(* PLC project SWPR1010_A0_1_29.project, CODESYS CODESYS V3.5 SP16 Patch 6 *)
(* stored: creationDateTime 2025-08-05T16:58:57.5396954, modificationDateTime 2025-08-05T16:58:31.4416113 *)

TYPE BOOL_T : STRUCT
  v : BOOL := TRUE;  (* Validation Bit *)
  e : BOOL := FALSE;  (* j1939 error bit *)
  na : BOOL := FALSE;  (* j1939 not available bit *)
  x : BOOL;  (* Value Bit *)
END_STRUCT;
END_TYPE

TYPE BYTE_T : STRUCT
  v : BOOL;  (* Validation Bit *)
  e : BOOL := FALSE;  (* j1939 error bit *)
  na : BOOL := FALSE;  (* j1939 not available bit *)
  x : BYTE;  (* Value Bit *)
  J1939 : BOOL;  (* J1939 *)
  RangeExcd : BOOL;  (* Range Exceeded *)
END_STRUCT;
END_TYPE

TYPE DWORD_T : STRUCT
  v : BOOL;  (* Validation Bit *)
  e : BOOL := FALSE;  (* j1939 error bit *)
  na : BOOL := FALSE;  (* j1939 not available bit *)
  x : DWORD;  (* Value Bit *)
  J1939 : BOOL;  (* J1939 *)
  RangeExcd : BOOL;  (* Range Exceeded *)
END_STRUCT;
END_TYPE

TYPE LREAL_T : STRUCT
  v : BOOL;  (* Validation Bit *)
  e : BOOL := FALSE;  (* j1939 error bit *)
  na : BOOL := FALSE;  (* j1939 not available bit *)
  x : LREAL;  (* Value Bit *)
  J1939 : BOOL;  (* J1939 *)
  RangeExcd : BOOL;  (* Range Exceeded *)
END_STRUCT;
END_TYPE

TYPE LWORD_T : STRUCT
  v : BOOL;  (* Validation Bit *)
  e : BOOL := FALSE;  (* j1939 error bit *)
  na : BOOL := FALSE;  (* j1939 not available bit *)
  x : LWORD;  (* Value Bit *)
  J1939 : BOOL;  (* J1939 *)
  RangeExcd : BOOL;  (* Range Exceeded *)
END_STRUCT;
END_TYPE

TYPE REAL_T : STRUCT
  v : BOOL;  (* Validation Bit *)
  e : BOOL := FALSE;  (* j1939 error bit *)
  na : BOOL := FALSE;  (* j1939 not available bit *)
  x : REAL;  (* Value Bit *)
  J1939 : BOOL;  (* J1939 *)
  RangeExcd : BOOL;  (* Range Exceeded *)
END_STRUCT;
END_TYPE

TYPE UDINT_T : STRUCT
  v : BOOL;  (* Validation Bit *)
  e : BOOL := FALSE;  (* j1939 error bit *)
  na : BOOL := FALSE;  (* j1939 not available bit *)
  x : UDINT;  (* Value Bit *)
  J1939 : BOOL;  (* J1939 *)
  RangeExcd : BOOL;  (* Range Exceeded *)
END_STRUCT;
END_TYPE

TYPE UINT_T : STRUCT
  v : BOOL;  (* Validation Bit *)
  e : BOOL := FALSE;  (* j1939 error bit *)
  na : BOOL := FALSE;  (* j1939 not available bit *)
  x : UINT;  (* Value Bit *)
  J1939 : BOOL;  (* J1939 *)
  RangeExcd : BOOL;  (* Range Exceeded *)
END_STRUCT;
END_TYPE

TYPE ULINT_T : STRUCT
  v : BOOL;  (* Validation Bit *)
  e : BOOL := FALSE;  (* j1939 error bit *)
  na : BOOL := FALSE;  (* j1939 not available bit *)
  x : ULINT;  (* Value Bit *)
  J1939 : BOOL;  (* J1939 *)
  RangeExcd : BOOL;  (* Range Exceeded *)
END_STRUCT;
END_TYPE

TYPE USINT_T : STRUCT
  v : BOOL;  (* Validation Bit *)
  e : BOOL := FALSE;  (* j1939 error bit *)
  na : BOOL := FALSE;  (* j1939 not available bit *)
  x : USINT;  (* Value Bit *)
  J1939 : BOOL;  (* J1939 *)
  RangeExcd : BOOL;  (* Range Exceeded *)
END_STRUCT;
END_TYPE

TYPE WORD_T : STRUCT
  v : BOOL;  (* Validation Bit *)
  e : BOOL := FALSE;  (* j1939 error bit *)
  na : BOOL := FALSE;  (* j1939 not available bit *)
  x : WORD;  (* Value Bit *)
  J1939 : BOOL;  (* J1939 *)
  RangeExcd : BOOL;  (* Range Exceeded *)
END_STRUCT;
END_TYPE

TYPE IIVD_T : STRUCT
  X_Param_Arr : Param_T;
  X_Spd_Max : REAL_T := (v := FALSE);  (* test *)
  S_ER_Com_ECU : BOOL_T := (v := FALSE);  (* ****************************************** MESSAGE: Haberlesme_Durumlari ID: 200 ****************************************** S_ER_Com_ECU/StartBit:0/Length:2/J1939:YES *)
  S_ER_Com_DWP_ICAN : BOOL_T := (v := FALSE);  (* S_ER_Com_DWP_ICAN/StartBit:2/Length:2/J1939:YES *)
  S_ER_Com_DWP_XCAN : BOOL_T := (v := FALSE);  (* S_ER_Com_DWP_XCAN/StartBit:4/Length:2/J1939:YES *)
  S_ER_Com_Str_Pmp : BOOL_T := (v := FALSE);  (* S_ER_Com_Str_Pmp/StartBit:6/Length:2/J1939:YES *)
  S_ER_Com_Fus_Chk_ID0 : BOOL_T := (v := FALSE);  (* S_ER_Com_Fus_Chk_ID0/StartBit:8/Length:2/J1939:YES *)
  S_ER_Com_Fus_Chk_ID1 : BOOL_T := (v := FALSE);  (* S_ER_Com_Fus_Chk_ID1/StartBit:10/Length:2/J1939:YES *)
  S_ER_Com_Fus_Chk_ID2 : BOOL_T := (v := FALSE);  (* S_ER_Com_Fus_Chk_ID2/StartBit:12/Length:2/J1939:YES *)
  S_ER_Com_ECAS : BOOL_T := (v := FALSE);  (* S_ER_Com_ECAS/StartBit:14/Length:2/J1939:YES *)
  S_ER_Com_Snd_Gen : BOOL_T := (v := FALSE);  (* S_ER_Com_Snd_Gen/StartBit:16/Length:2/J1939:YES *)
  S_ER_Com_DCAN : BOOL_T := (v := FALSE);  (* S_ER_Com_DCAN/StartBit:18/Length:2/J1939:YES *)
  S_ER_Com_Node1 : BOOL_T := (v := FALSE);  (* S_ER_Com_Node1/StartBit:24/Length:2/J1939:YES *)
  S_ER_Com_Node2 : BOOL_T := (v := FALSE);  (* S_ER_Com_Node2/StartBit:26/Length:2/J1939:YES *)
  S_ER_Com_Node3 : BOOL_T := (v := FALSE);  (* S_ER_Com_Node3/StartBit:28/Length:2/J1939:YES *)
  S_ER_Com_Node4 : BOOL_T := (v := FALSE);  (* S_ER_Com_Node4/StartBit:30/Length:2/J1939:YES *)
  S_ER_Com_Node5 : BOOL_T := (v := FALSE);  (* S_ER_Com_Node5/StartBit:32/Length:2/J1939:YES *)
  S_ER_Com_Node6 : BOOL_T := (v := FALSE);  (* S_ER_Com_Node6/StartBit:34/Length:2/J1939:YES *)
  S_ER_Com_Node8 : BOOL_T := (v := FALSE);  (* S_ER_Com_Node8/StartBit:38/Length:2/J1939:YES *)
  S_ER_Com_Dr1 : BOOL_T := (v := FALSE);  (* S_ER_Com_Dr1/StartBit:40/Length:2/J1939:YES *)
  S_ER_Com_Dr2 : BOOL_T := (v := FALSE);  (* S_ER_Com_Dr2/StartBit:42/Length:2/J1939:YES *)
  S_ER_Com_Dr3 : BOOL_T := (v := FALSE);  (* S_ER_Com_Dr3/StartBit:44/Length:2/J1939:YES *)
  S_ER_Com_Dr4 : BOOL_T := (v := FALSE);  (* S_ER_Com_Dr4/StartBit:46/Length:2/J1939:YES *)
  S_ER_Com_Dr5 : BOOL_T := (v := FALSE);  (* S_ER_Com_Dr5/StartBit:48/Length:2/J1939:YES *)
  S_ER_Com_Dr6 : BOOL_T := (v := FALSE);  (* S_ER_Com_Dr6/StartBit:50/Length:2/J1939:YES *)
  S_ER_Com_Dr7 : BOOL_T := (v := FALSE);  (* S_ER_Com_Dr7/StartBit:52/Length:2/J1939:YES *)
  S_ER_Com_Dr8 : BOOL_T := (v := FALSE);  (* S_ER_Com_Dr8/StartBit:54/Length:2/J1939:YES *)
  S_ER_Com_Dr9 : BOOL_T := (v := FALSE);  (* S_ER_Com_Dr9/StartBit:56/Length:2/J1939:YES *)
  S_Warn_Knl_Mn_Cond : BOOL_T := (v := FALSE);  (* S_Warn_Knl_Mn_Cond/StartBit:58/Length:2/J1939:YES *)
  S_ER_Lmp_Oc : BOOL_T := (v := FALSE);  (* S_ER_Lmp_Oc/StartBit:60/Length:2/J1939:YES *)
  S_ER_Mir_Windw_Heat_En : BOOL_T := (v := FALSE);  (* S_ER_Mir_Windw_Heat_En/StartBit:62/Length:2/J1939:YES *)
  W_Str_Pmp_Spd : REAL_T := (v := FALSE);  (* ****************************************** MESSAGE: Direksiyon_Pompasi_Analog ID: 210 ****************************************** W_Str_Pmp_Spd/StartBit:0/Length:16/J1939:YES *)
  X_Str_Pmp_Spd : REAL_T := (v := FALSE);  (* X_Str_Pmp_Spd/StartBit:16/Length:16/J1939:YES *)
  X_P_Str_Pmp : REAL_T := (v := FALSE);  (* X_P_Str_Pmp/StartBit:32/Length:16/J1939:YES *)
  X_I_Str_Pmp : REAL_T := (v := FALSE);  (* X_I_Str_Pmp/StartBit:48/Length:9/J1939:NO *)
  C_Str_Pmp_En : BOOL_T := (v := FALSE);  (* ****************************************** MESSAGE: Direksiyon_Pompasi_Durum ID: 211 ****************************************** C_Str_Pmp_En/StartBit:0/Length:2/J1939:YES *)
  S_Str_Pmp_Em_Run_FOC : BOOL_T := (v := FALSE);  (* S_Str_Pmp_Em_Run_FOC/StartBit:2/Length:2/J1939:YES *)
  S_Str_Pmp_Em_Run_Slp : BOOL_T := (v := FALSE);  (* S_Str_Pmp_Em_Run_Slp/StartBit:4/Length:2/J1939:YES *)
  S_ER_Str_Pmp : BOOL_T := (v := FALSE);  (* S_ER_Str_Pmp/StartBit:6/Length:2/J1939:YES *)
  S_Str_Pmp_Run : BOOL_T := (v := FALSE);  (* S_Str_Pmp_Run/StartBit:8/Length:2/J1939:YES *)
  X_T_Str_Pmp_Mot : REAL_T := (v := FALSE);  (* X_T_Str_Pmp_Mot/StartBit:16/Length:8/J1939:YES *)
  X_T_Str_Pmp_Inver : REAL_T := (v := FALSE);  (* X_T_Str_Pmp_Inver/StartBit:24/Length:8/J1939:YES *)
  X_Mot_Load_Str_Pmp : REAL_T := (v := FALSE);  (* X_Mot_Load_Str_Pmp/StartBit:32/Length:8/J1939:YES *)
  X_T_Air_Cmp : REAL_T := (v := FALSE);  (* X_T_Air_Cmp/StartBit:48/Length:8/J1939:YES *)
  S_ER_Air_Cmp_Tmp : BOOL_T := (v := FALSE);  (* S_ER_Air_Cmp_Tmp/StartBit:56/Length:2/J1939:YES *)
  S_Air_Cmp_Filt_Warn_Actv : BOOL_T := (v := FALSE);  (* S_Air_Cmp_Filt_Warn_Actv/StartBit:58/Length:2/J1939:YES *)
  S_Hld_Brk_Byp : BOOL_T := (v := FALSE);  (* ****************************************** MESSAGE: Arac_Durumlari ID: 220 ****************************************** S_Hld_Brk_Byp/StartBit:0/Length:2/J1939:YES *)
  S_Hld_Brk_Req : BOOL_T := (v := FALSE);  (* S_Hld_Brk_Req/StartBit:2/Length:2/J1939:YES *)
  S_Hld_Brk_Actv : BOOL_T := (v := FALSE);  (* S_Hld_Brk_Actv/StartBit:4/Length:2/J1939:YES *)
  S_Aut_Lub_Oil_Lv_Lo : BOOL_T := (v := FALSE);  (* S_Aut_Lub_Oil_Lv_Lo/StartBit:6/Length:2/J1939:YES *)
  S_ECAS_Dwn_Req : BOOL_T := (v := FALSE);  (* S_ECAS_Dwn_Req/StartBit:8/Length:2/J1939:YES *)
  S_ECAS_Up_Req : BOOL_T := (v := FALSE);  (* S_ECAS_Up_Req/StartBit:10/Length:2/J1939:YES *)
  S_ECAS_Pos_Down : BOOL_T := (v := FALSE);  (* S_ECAS_Pos_Down/StartBit:12/Length:2/J1939:YES *)
  S_ECAS_Pos_Up : BOOL_T := (v := FALSE);  (* S_ECAS_Pos_Up/StartBit:14/Length:2/J1939:YES *)
  S_Knl_Req : BOOL_T := (v := FALSE);  (* S_Knl_Req/StartBit:16/Length:2/J1939:YES *)
  S_Knl_Actv : BOOL_T := (v := FALSE);  (* S_Knl_Actv/StartBit:18/Length:2/J1939:YES *)
  S_Fwd_Gear : BOOL_T := (v := FALSE);  (* S_Fwd_Gear/StartBit:20/Length:2/J1939:YES *)
  S_Bwd_Gear : BOOL_T := (v := FALSE);  (* S_Bwd_Gear/StartBit:22/Length:2/J1939:YES *)
  S_Vh_Actv_Key_Lv1 : BOOL_T := (v := FALSE);  (* S_Vh_Actv_Key_Lv1/StartBit:24/Length:2/J1939:YES *)
  S_Vh_Actv_Key_Lv2 : BOOL_T := (v := FALSE);  (* S_Vh_Actv_Key_Lv2/StartBit:26/Length:2/J1939:YES *)
  S_Vh_Actv_Key_Lv3 : BOOL_T := (v := FALSE);  (* S_Vh_Actv_Key_Lv3/StartBit:28/Length:2/J1939:YES *)
  S_Brk_Park : BOOL_T := (v := FALSE);  (* S_Brk_Park/StartBit:30/Length:2/J1939:YES *)
  Z_Ret_Lv : BYTE_T := (v := FALSE);  (* Z_Ret_Lv/StartBit:32/Length:4/J1939:YES *)
  S_Aut_Lub_Actv : BOOL_T := (v := FALSE);  (* S_Aut_Lub_Actv/StartBit:36/Length:2/J1939:YES *)
  S_ER_Aut_Lub_Snsr : BOOL_T := (v := FALSE);  (* S_ER_Aut_Lub_Snsr/StartBit:38/Length:2/J1939:YES *)
  S_Bat_Mod_Btn : BOOL_T := (v := FALSE);  (* S_Bat_Mod_Btn/StartBit:42/Length:2/J1939:YES *)
  S_Elec_Mod_Btn : BOOL_T := (v := FALSE);  (* S_Elec_Mod_Btn/StartBit:44/Length:2/J1939:YES *)
  S_Bwd_Lft_Chrg_Btn : BOOL_T := (v := FALSE);  (* S_Bwd_Lft_Chrg_Btn/StartBit:12/Length:2/J1939:YES *)
  S_Bwd_Lft_Chrg_Em_Stop_Swc1 : BOOL_T := (v := FALSE);  (* S_Bwd_Lft_Chrg_Em_Stop_Swc1/StartBit:14/Length:2/J1939:YES *)
  S_Bwd_Lft_Chrg_Em_Stop_Swc2 : BOOL_T := (v := FALSE);  (* S_Bwd_Lft_Chrg_Em_Stop_Swc2/StartBit:16/Length:2/J1939:YES *)
  Z_Config_Clu : BYTE_T := (v := FALSE);  (* Z_Config_Clu/StartBit:56/Length:8/J1939:YES *)
  X_Axl1_Brk_Ling_1 : REAL_T := (v := FALSE);  (* ****************************************** MESSAGE: Fren_balata_durumlari ID: 221 ****************************************** X_Axl1_Brk_Ling_1/StartBit:0/Length:8/J1939:YES *)
  X_Axl1_Brk_Ling_2 : REAL_T := (v := FALSE);  (* X_Axl1_Brk_Ling_2/StartBit:8/Length:8/J1939:YES *)
  X_Axl2_Brk_Ling_1 : REAL_T := (v := FALSE);  (* X_Axl2_Brk_Ling_1/StartBit:16/Length:8/J1939:YES *)
  X_Axl2_Brk_Ling_2 : REAL_T := (v := FALSE);  (* X_Axl2_Brk_Ling_2/StartBit:24/Length:8/J1939:YES *)
  X_Axl3_Brk_Ling_1 : REAL_T := (v := FALSE);  (* X_Axl3_Brk_Ling_1/StartBit:32/Length:8/J1939:YES *)
  X_Axl3_Brk_Ling_2 : REAL_T := (v := FALSE);  (* X_Axl3_Brk_Ling_2/StartBit:40/Length:8/J1939:YES *)
  X_Axl4_Brk_Ling_1 : REAL_T := (v := FALSE);  (* X_Axl4_Brk_Ling_1/StartBit:48/Length:8/J1939:YES *)
  X_Axl4_Brk_Ling_2 : REAL_T := (v := FALSE);  (* X_Axl4_Brk_Ling_2/StartBit:56/Length:8/J1939:YES *)
  S_ER_Not_Ins_Pr_Sns_Frnt_Brk : BOOL_T := (v := FALSE);  (* ****************************************** MESSAGE: Fren_Basinclari ID: 222 ****************************************** S_ER_Not_Ins_Pr_Sns_Frnt_Brk/StartBit:0/Length:2/J1939:YES *)
  S_ER_Not_Ins_Pr_Sns_Bwd_Brk : BOOL_T := (v := FALSE);  (* S_ER_Not_Ins_Pr_Sns_Bwd_Brk/StartBit:2/Length:2/J1939:YES *)
  S_ER_Not_Ins_Pr_Snsr_Prk_Brk : BOOL_T := (v := FALSE);  (* S_ER_Not_Ins_Pr_Snsr_Prk_Brk/StartBit:4/Length:2/J1939:YES *)
  S_ER_Not_Ins_Pr_Sns_Susp_Rr : BOOL_T := (v := FALSE);  (* S_ER_Not_Ins_Pr_Sns_Susp/StartBit:6/Length:2/J1939:YES *)
  S_ER_Not_Ins_Pr_Sns_Susp_Frnt : BOOL_T := (v := FALSE);  (* S_ER_Not_Ins_Pr_Sns_Susp_Frnt/StartBit:8/Length:2/J1939:YES *)
  S_ER_Brk_Lnng : BOOL_T := (v := FALSE);  (* S_ER_Brk_Lnng/StartBit:8/Length:2/J1939:YES *)
  S_ER_Pin_Pr_Air : BOOL_T := (v := FALSE);  (* S_ER_Pin_Pr_Air/StartBit:12/Length:2/J1939:YES *)
  X_Pr_Air_Tank_Brk_Bwd : REAL_T := (v := FALSE);  (* X_Pr_Air_Tank_Brk_Bwd/StartBit:16/Length:8/J1939:YES *)
  X_Pr_Air_Tank_Brk_Frnt : REAL_T := (v := FALSE);  (* X_Pr_Air_Tank_Brk_Frnt/StartBit:24/Length:8/J1939:YES *)
  X_Pr_Air_Tank_Brk_Prk : REAL_T := (v := FALSE);  (* X_Pr_Air_Tank_Brk_Prk/StartBit:32/Length:8/J1939:YES *)
  X_Pr_Air_Tank_Susp_Rr : REAL_T := (v := FALSE);  (* X_Pr_Air_Tank_Susp_Rr/StartBit:40/Length:8/J1939:YES *)
  X_Pr_Air_Tank_Susp_Frnt : REAL_T := (v := FALSE);  (* X_Pr_Air_Tank_Susp_Frnt/StartBit:48/Length:8/J1939:YES *)
  X_Pr_Axl1_Wh1 : REAL_T := (v := FALSE);  (* ****************************************** MESSAGE: Lastik_Basinclari_1 ID: 223 ****************************************** X_Pr_Axl1_Wh1/StartBit:0/Length:8/J1939:YES *)
  X_Pr_Axl1_Wh2 : REAL_T := (v := FALSE);  (* X_Pr_Axl1_Wh2/StartBit:8/Length:8/J1939:YES *)
  X_Pr_Axl2_Wh1 : REAL_T := (v := FALSE);  (* X_Pr_Axl2_Wh1/StartBit:16/Length:8/J1939:YES *)
  X_Pr_Axl2_Wh2 : REAL_T := (v := FALSE);  (* X_Pr_Axl2_Wh2/StartBit:24/Length:8/J1939:YES *)
  X_Pr_Axl2_Wh3 : REAL_T := (v := FALSE);  (* X_Pr_Axl2_Wh3/StartBit:32/Length:8/J1939:YES *)
  X_Pr_Axl2_Wh4 : REAL_T := (v := FALSE);  (* X_Pr_Axl2_Wh4/StartBit:40/Length:8/J1939:YES *)
  X_Pr_Axl3_Wh1 : REAL_T := (v := FALSE);  (* ****************************************** MESSAGE: Lastik_Basinclari_2 ID: 224 ****************************************** X_Pr_Axl3_Wh1/StartBit:0/Length:8/J1939:YES *)
  X_Pr_Axl3_Wh2 : REAL_T := (v := FALSE);  (* X_Pr_Axl3_Wh2/StartBit:8/Length:8/J1939:YES *)
  X_Pr_Axl3_Wh3 : REAL_T := (v := FALSE);  (* X_Pr_Axl3_Wh3/StartBit:16/Length:8/J1939:YES *)
  X_Pr_Axl3_Wh4 : REAL_T := (v := FALSE);  (* X_Pr_Axl3_Wh4/StartBit:24/Length:8/J1939:YES *)
  X_Pr_Axl4_Wh1 : REAL_T := (v := FALSE);  (* X_Pr_Axl4_Wh1/StartBit:32/Length:8/J1939:YES *)
  X_Pr_Axl4_Wh2 : REAL_T := (v := FALSE);  (* X_Pr_Axl4_Wh2/StartBit:40/Length:8/J1939:YES *)
  X_Pr_Axl4_Wh3 : REAL_T := (v := FALSE);  (* X_Pr_Axl4_Wh3/StartBit:48/Length:8/J1939:YES *)
  X_Pr_Axl4_Wh4 : REAL_T := (v := FALSE);  (* X_Pr_Axl4_Wh4/StartBit:56/Length:8/J1939:YES *)
  S_Cvr_Op_Dr1_Ext : BOOL_T := (v := FALSE);  (* ****************************************** MESSAGE: Arac_Bilgilendirme ID: 225 ****************************************** S_Cvr_Op_Dr1_Ext/StartBit:0/Length:2/J1939:YES *)
  S_Cvr_Op_Lic : BOOL_T := (v := FALSE);  (* S_Cvr_Op_Lic/StartBit:2/Length:2/J1939:YES *)
  S_Cvr_Op_Bat_Room : BOOL_T := (v := FALSE);  (* S_Cvr_Op_Bat_Room/StartBit:4/Length:2/J1939:YES *)
  S_Cvr_Op_Mot : BOOL_T := (v := FALSE);  (* S_Cvr_Op_Mot/StartBit:10/Length:2/J1939:YES *)
  S_Cvr_Op_Bwd_Lft_Chrg : BOOL_T := (v := FALSE);  (* S_Cvr_Op_Bwd_Lft_Chrg/StartBit:12/Length:2/J1939:YES *)
  S_Cvr_Op_24V_Chrg_Plg : BOOL_T := (v := FALSE);  (* S_Cvr_Op_24V_Chrg_Plg/StartBit:14/Length:2/J1939:YES *)
  S_Cvr_Op_Bwd : BOOL_T := (v := FALSE);  (* S_Cvr_Op_Bwd/StartBit:16/Length:2/J1939:YES *)
  S_Rp_Op : BOOL_T := (v := FALSE);  (* S_Rp_Op/StartBit:18/Length:2/J1939:YES *)
  S_Cvr_Op_Bwd_Mnt_Pnl : BOOL_T := (v := FALSE);  (* S_Cvr_Op_Bwd_Mnt_Pnl/StartBit:20/Length:2/J1939:YES *)
  S_Cvr_Op_Frnt_Mnt_Pnl : BOOL_T := (v := FALSE);  (* S_Cvr_Op_Frnt_Mnt_Pnl/StartBit:22/Length:2/J1939:YES *)
  S_ER_Rp_Op_Unauth : BOOL_T := (v := FALSE);  (* S_ER_Rp_Op_Unauth/StartBit:30/Length:2/J1939:YES *)
  S_ER_Fi_Bat_Room : BOOL_T := (v := FALSE);  (* S_ER_Fi_Bat_Room/StartBit:32/Length:2/J1939:YES *)
  S_ER_Not_Ins_Fi_Sens_Bat_Room : BOOL_T := (v := FALSE);  (* S_ER_Not_Ins_Fi_Sens_Bat_Room/StartBit:34/Length:2/J1939:YES *)
  S_ER_Fi_Frnt_Pnl : BOOL_T := (v := FALSE);  (* S_ER_Fi_Frnt_Pnl/StartBit:36/Length:2/J1939:YES *)
  S_ER_Not_Ins_Fi_Snsr_Frnt_Pnl : BOOL_T := (v := FALSE);  (* S_ER_Not_Ins_Fi_Snsr_Frnt_Pnl/StartBit:38/Length:2/J1939:YES *)
  S_ER_Fi_Drv_Mot : BOOL_T := (v := FALSE);  (* S_ER_Fi_Drv_Mot/StartBit:40/Length:2/J1939:YES *)
  S_ER_Not_Ins_Fi_Snsr_Drv_Mot : BOOL_T := (v := FALSE);  (* S_ER_Not_Ins_Fi_Snsr_Drv_Mot/StartBit:42/Length:2/J1939:YES *)
  S_ER_Fi_Bwd_Pnl : BOOL_T := (v := FALSE);  (* S_ER_Fi_Bwd_Pnl/StartBit:44/Length:2/J1939:YES *)
  S_ER_Not_Ins_Fi_Snsr_Bwd_Pnl : BOOL_T := (v := FALSE);  (* S_ER_Not_Ins_Fi_Snsr_Bwd_Pnl/StartBit:46/Length:2/J1939:YES *)
  S_ER_Fi_Eng_Room : BOOL_T := (v := FALSE);  (* S_ER_Fi_Eng_Room/StartBit:48/Length:2/J1939:YES *)
  S_ER_Not_Ins_Fi_Sns_Eng_Room : BOOL_T := (v := FALSE);  (* S_ER_Not_Ins_Fi_Sns_Eng_Room/StartBit:50/Length:2/J1939:YES *)
  X_Psng_No : REAL_T := (v := FALSE);  (* ****************************************** MESSAGE: Arac_Kritik_Uyarilari ID: 226 ****************************************** X_Psng_No/StartBit:0/Length:8/J1939:YES *)
  X_Wgt_Axle : REAL_T := (v := FALSE);  (* X_Wgt_Axle/StartBit:8/Length:16/J1939:YES *)
  C_Err_Pg_Dn : BOOL_T := (v := FALSE);  (* C_Err_Pg_Dn/StartBit:24/Length:2/J1939:YES *)
  C_Err_Pg_Up : BOOL_T := (v := FALSE);  (* C_Err_Pg_Up/StartBit:26/Length:2/J1939:YES *)
  C_Rst_Trip : BOOL_T := (v := FALSE);  (* C_Rst_Trip/StartBit:28/Length:2/J1939:YES *)
  S_Drug_Alch_Ctrl : BOOL_T := (v := FALSE);  (* S_Drug_Alch_Ctrl/StartBit:32/Length:2/J1939:YES *)
  S_Drug_Alch_Warn : BOOL_T := (v := FALSE);  (* S_Drug_Alch_Warn/StartBit:34/Length:2/J1939:YES *)
  S_Prheat_Tk_Lv_Lo : BOOL_T := (v := FALSE);  (* C_Flr_Heat_Off/StartBit:36/Length:2/J1939:YES *)
  S_ER_Wpr_Wtr_Lv : BOOL_T := (v := FALSE);  (* S_ER_Wpr_Wtr_Lv/StartBit:40/Length:2/J1939:YES *)
  S_Sfty_Belt_Ins : BOOL_T := (v := FALSE);  (* S_Sfty_Belt_Ins/StartBit:42/Length:2/J1939:YES *)
  C_Pnt_Up : BOOL_T := (v := FALSE);  (* C_Pnt_Up/StartBit:44/Length:2/J1939:YES *)
  C_Pnt_Dn : BOOL_T := (v := FALSE);  (* C_Pnt_Dn/StartBit:46/Length:2/J1939:YES *)
  S_Drv_Seat_Pre_Snsr : BOOL_T := (v := FALSE);  (* S_Drv_Seat_Pre_Snsr/StartBit:48/Length:2/J1939:YES *)
  S_Inc_Acc : BOOL_T := (v := FALSE);  (* S_Inc_Acc/StartBit:56/Length:2/J1939:YES *)
  S_Inc_Stop : BOOL_T := (v := FALSE);  (* S_Inc_Stop/StartBit:58/Length:2/J1939:YES *)
  S_Er_Tire_Pres : BOOL_T := (v := FALSE);  (* S_Er_Tire_Pres/StartBit:60/Length:2/J1939:YES *)
  Z_Dr1_Err_Fram_1 : BYTE_T := (v := FALSE);  (* ****************************************** MESSAGE: Kapi_Hatalari_1 ID: 230 ****************************************** Z_Dr1_Err_Fram_1/StartBit:0/Length:8/J1939:YES *)
  Z_Dr1_Err_Fram_2 : BYTE_T := (v := FALSE);  (* Z_Dr1_Err_Fram_2/StartBit:8/Length:8/J1939:YES *)
  Z_Dr1_Err_Fram_3 : BYTE_T := (v := FALSE);  (* Z_Dr1_Err_Fram_3/StartBit:16/Length:8/J1939:YES *)
  Z_Dr2_Err_Fram_1 : BYTE_T := (v := FALSE);  (* Z_Dr2_Err_Fram_1/StartBit:32/Length:8/J1939:YES *)
  Z_Dr2_Err_Fram_2 : BYTE_T := (v := FALSE);  (* Z_Dr2_Err_Fram_2/StartBit:40/Length:8/J1939:YES *)
  Z_Dr2_Err_Fram_3 : BYTE_T := (v := FALSE);  (* Z_Dr2_Err_Fram_3/StartBit:48/Length:8/J1939:YES *)
  Z_Dr3_Err_Fram_1 : BYTE_T := (v := FALSE);  (* ****************************************** MESSAGE: Kapi_Hatalari_2 ID: 231 ****************************************** Z_Dr3_Err_Fram_1/StartBit:0/Length:8/J1939:YES *)
  Z_Dr3_Err_Fram_2 : BYTE_T := (v := FALSE);  (* Z_Dr3_Err_Fram_2/StartBit:8/Length:8/J1939:YES *)
  Z_Dr3_Err_Fram_3 : BYTE_T := (v := FALSE);  (* Z_Dr3_Err_Fram_3/StartBit:16/Length:8/J1939:YES *)
  Z_Dr4_Err_Fram_1 : BYTE_T := (v := FALSE);  (* Z_Dr4_Err_Fram_1/StartBit:32/Length:8/J1939:YES *)
  Z_Dr4_Err_Fram_2 : BYTE_T := (v := FALSE);  (* Z_Dr4_Err_Fram_2/StartBit:40/Length:8/J1939:YES *)
  Z_Dr4_Err_Fram_3 : BYTE_T := (v := FALSE);  (* Z_Dr4_Err_Fram_3/StartBit:48/Length:8/J1939:YES *)
  Z_Dr5_Err_Fram_1 : BYTE_T := (v := FALSE);  (* ****************************************** MESSAGE: Kapi_Hatalari_3 ID: 232 ****************************************** Z_Dr5_Err_Fram_1/StartBit:0/Length:8/J1939:YES *)
  Z_Dr5_Err_Fram_2 : BYTE_T := (v := FALSE);  (* Z_Dr5_Err_Fram_2/StartBit:8/Length:8/J1939:YES *)
  Z_Dr5_Err_Fram_3 : BYTE_T := (v := FALSE);  (* Z_Dr5_Err_Fram_3/StartBit:16/Length:8/J1939:YES *)
  Z_Dr6_Err_Fram_1 : BYTE_T := (v := FALSE);  (* Z_Dr6_Err_Fram_1/StartBit:32/Length:8/J1939:YES *)
  Z_Dr6_Err_Fram_2 : BYTE_T := (v := FALSE);  (* Z_Dr6_Err_Fram_2/StartBit:40/Length:8/J1939:YES *)
  Z_Dr6_Err_Fram_3 : BYTE_T := (v := FALSE);  (* Z_Dr6_Err_Fram_3/StartBit:48/Length:8/J1939:YES *)
  Z_Dr7_Err_Fram_1 : BYTE_T := (v := FALSE);  (* ****************************************** MESSAGE: Kapi_Hatalari_4 ID: 233 ****************************************** Z_Dr7_Err_Fram_1/StartBit:0/Length:8/J1939:YES *)
  Z_Dr7_Err_Fram_2 : BYTE_T := (v := FALSE);  (* Z_Dr7_Err_Fram_2/StartBit:8/Length:8/J1939:YES *)
  Z_Dr7_Err_Fram_3 : BYTE_T := (v := FALSE);  (* Z_Dr7_Err_Fram_3/StartBit:16/Length:8/J1939:YES *)
  Z_Dr8_Err_Fram_1 : BYTE_T := (v := FALSE);  (* Z_Dr8_Err_Fram_1/StartBit:32/Length:8/J1939:YES *)
  Z_Dr8_Err_Fram_2 : BYTE_T := (v := FALSE);  (* Z_Dr8_Err_Fram_2/StartBit:40/Length:8/J1939:YES *)
  Z_Dr8_Err_Fram_3 : BYTE_T := (v := FALSE);  (* Z_Dr8_Err_Fram_3/StartBit:48/Length:8/J1939:YES *)
  Z_Dr9_Err_Fram_1 : BYTE_T := (v := FALSE);  (* ****************************************** MESSAGE: Kapi_Hatalari_5 ID: 234 ****************************************** Z_Dr9_Err_Fram_1/StartBit:0/Length:8/J1939:YES *)
  Z_Dr9_Err_Fram_2 : BYTE_T := (v := FALSE);  (* Z_Dr9_Err_Fram_2/StartBit:8/Length:8/J1939:YES *)
  Z_Dr9_Err_Fram_3 : BYTE_T := (v := FALSE);  (* Z_Dr9_Err_Fram_3/StartBit:16/Length:8/J1939:YES *)
  S_Dr1_Rhs_Leaf_Opng : BOOL_T := (v := FALSE);  (* ****************************************** MESSAGE: Kapi_Durum_1 ID: 235 ****************************************** S_Dr1_Rhs_Leaf_Opng/StartBit:0/Length:2/J1939:YES *)
  S_Dr1_Rhs_Leaf_Clng : BOOL_T := (v := FALSE);  (* S_Dr1_Rhs_Leaf_Clng/StartBit:2/Length:2/J1939:YES *)
  S_Dr1_Rhs_Leaf_Op : BOOL_T := (v := FALSE);  (* S_Dr1_Rhs_Leaf_Op/StartBit:4/Length:2/J1939:YES *)
  S_Dr1_Rhs_Leaf_Cl : BOOL_T := (v := FALSE);  (* S_Dr1_Rhs_Leaf_Cl/StartBit:6/Length:2/J1939:YES *)
  S_Dr1_Rhs_Leaf_Obs : BOOL_T := (v := FALSE);  (* S_Dr1_Rhs_Leaf_Obs/StartBit:8/Length:2/J1939:YES *)
  S_Dr1_Lft_Leaf_Opng : BOOL_T := (v := FALSE);  (* S_Dr1_Lft_Leaf_Opng/StartBit:10/Length:2/J1939:YES *)
  S_Dr1_Lft_Leaf_Clng : BOOL_T := (v := FALSE);  (* S_Dr1_Lft_Leaf_Clng/StartBit:12/Length:2/J1939:YES *)
  S_Dr1_Lft_Leaf_Op : BOOL_T := (v := FALSE);  (* S_Dr1_Lft_Leaf_Op/StartBit:14/Length:2/J1939:YES *)
  S_Dr1_Lft_Leaf_Cl : BOOL_T := (v := FALSE);  (* S_Dr1_Lft_Leaf_Cl/StartBit:16/Length:2/J1939:YES *)
  S_Dr1_Lft_Leaf_Obs : BOOL_T := (v := FALSE);  (* S_Dr1_Lft_Leaf_Obs/StartBit:18/Length:2/J1939:YES *)
  S_Dr1_Em_Swc : BOOL_T := (v := FALSE);  (* S_Dr1_Em_Swc/StartBit:20/Length:2/J1939:YES *)
  S_Dr2_Opng : BOOL_T := (v := FALSE);  (* S_Dr2_Opng/StartBit:24/Length:2/J1939:YES *)
  S_Dr2_Clng : BOOL_T := (v := FALSE);  (* S_Dr2_Clng/StartBit:26/Length:2/J1939:YES *)
  S_Dr2_Op : BOOL_T := (v := FALSE);  (* S_Dr2_Op/StartBit:28/Length:2/J1939:YES *)
  S_Dr2_Cl : BOOL_T := (v := FALSE);  (* S_Dr2_Cl/StartBit:30/Length:2/J1939:YES *)
  S_Dr2_Obs : BOOL_T := (v := FALSE);  (* S_Dr2_Obs/StartBit:32/Length:2/J1939:YES *)
  S_Dr2_Em_Swc : BOOL_T := (v := FALSE);  (* S_Dr2_Em_Swc/StartBit:34/Length:2/J1939:YES *)
  S_Dr3_Opng : BOOL_T := (v := FALSE);  (* S_Dr3_Opng/StartBit:40/Length:2/J1939:YES *)
  S_Dr3_Clng : BOOL_T := (v := FALSE);  (* S_Dr3_Clng/StartBit:42/Length:2/J1939:YES *)
  S_Dr3_Op : BOOL_T := (v := FALSE);  (* S_Dr3_Op/StartBit:44/Length:2/J1939:YES *)
  S_Dr3_Cl : BOOL_T := (v := FALSE);  (* S_Dr3_Cl/StartBit:46/Length:2/J1939:YES *)
  S_Dr3_Obs : BOOL_T := (v := FALSE);  (* S_Dr3_Obs/StartBit:48/Length:2/J1939:YES *)
  S_Dr3_Em_Swc : BOOL_T := (v := FALSE);  (* S_Dr3_Em_Swc/StartBit:50/Length:2/J1939:YES *)
  S_Dr4_Opng : BOOL_T := (v := FALSE);  (* ****************************************** MESSAGE: Kapi_Durum_2 ID: 237 ****************************************** S_Dr4_Opng/StartBit:0/Length:2/J1939:YES *)
  S_Dr4_Clng : BOOL_T := (v := FALSE);  (* S_Dr4_Clng/StartBit:2/Length:2/J1939:YES *)
  S_Dr4_Op : BOOL_T := (v := FALSE);  (* S_Dr4_Op/StartBit:4/Length:2/J1939:YES *)
  S_Dr4_Cl : BOOL_T := (v := FALSE);  (* S_Dr4_Cl/StartBit:6/Length:2/J1939:YES *)
  S_Dr4_Obs : BOOL_T := (v := FALSE);  (* S_Dr4_Obs/StartBit:8/Length:2/J1939:YES *)
  S_Dr4_Em_Swc : BOOL_T := (v := FALSE);  (* S_Dr4_Em_Swc/StartBit:10/Length:2/J1939:YES *)
  S_Dr5_Opng : BOOL_T := (v := FALSE);  (* S_Dr5_Opng/StartBit:16/Length:2/J1939:YES *)
  S_Dr5_Clng : BOOL_T := (v := FALSE);  (* S_Dr5_Clng/StartBit:18/Length:2/J1939:YES *)
  S_Dr5_Op : BOOL_T := (v := FALSE);  (* S_Dr5_Op/StartBit:20/Length:2/J1939:YES *)
  S_Dr5_Cl : BOOL_T := (v := FALSE);  (* S_Dr5_Cl/StartBit:22/Length:2/J1939:YES *)
  S_Dr5_Obs : BOOL_T := (v := FALSE);  (* S_Dr5_Obs/StartBit:24/Length:2/J1939:YES *)
  S_Dr5_Em_Swc : BOOL_T := (v := FALSE);  (* S_Dr5_Em_Swc/StartBit:26/Length:2/J1939:YES *)
  S_Dr6_Opng : BOOL_T := (v := FALSE);  (* S_Dr6_Opng/StartBit:32/Length:2/J1939:YES *)
  S_Dr6_Clng : BOOL_T := (v := FALSE);  (* S_Dr6_Clng/StartBit:34/Length:2/J1939:YES *)
  S_Dr6_Op : BOOL_T := (v := FALSE);  (* S_Dr6_Op/StartBit:36/Length:2/J1939:YES *)
  S_Dr6_Cl : BOOL_T := (v := FALSE);  (* S_Dr6_Cl/StartBit:38/Length:2/J1939:YES *)
  S_Dr6_Obs : BOOL_T := (v := FALSE);  (* S_Dr6_Obs/StartBit:40/Length:2/J1939:YES *)
  S_Dr6_Em_Swc : BOOL_T := (v := FALSE);  (* S_Dr6_Em_Swc/StartBit:42/Length:2/J1939:YES *)
  S_Dr7_Opng : BOOL_T := (v := FALSE);  (* ****************************************** MESSAGE: Kapi_Durum_3 ID: 238 ****************************************** S_Dr7_Opng/StartBit:0/Length:2/J1939:YES *)
  S_Dr7_Clng : BOOL_T := (v := FALSE);  (* S_Dr7_Clng/StartBit:2/Length:2/J1939:YES *)
  S_Dr7_Op : BOOL_T := (v := FALSE);  (* S_Dr7_Op/StartBit:4/Length:2/J1939:YES *)
  S_Dr7_Cl : BOOL_T := (v := FALSE);  (* S_Dr7_Cl/StartBit:6/Length:2/J1939:YES *)
  S_Dr7_Obs : BOOL_T := (v := FALSE);  (* S_Dr7_Obs/StartBit:8/Length:2/J1939:YES *)
  S_Dr7_Em_Swc : BOOL_T := (v := FALSE);  (* S_Dr7_Em_Swc/StartBit:10/Length:2/J1939:YES *)
  S_Dr8_Opng : BOOL_T := (v := FALSE);  (* S_Dr8_Opng/StartBit:16/Length:2/J1939:YES *)
  S_Dr8_Clng : BOOL_T := (v := FALSE);  (* S_Dr8_Clng/StartBit:18/Length:2/J1939:YES *)
  S_Dr8_Op : BOOL_T := (v := FALSE);  (* S_Dr8_Op/StartBit:20/Length:2/J1939:YES *)
  S_Dr8_Cl : BOOL_T := (v := FALSE);  (* S_Dr8_Cl/StartBit:22/Length:2/J1939:YES *)
  S_Dr8_Obs : BOOL_T := (v := FALSE);  (* S_Dr8_Obs/StartBit:24/Length:2/J1939:YES *)
  S_Dr8_Em_Swc : BOOL_T := (v := FALSE);  (* S_Dr8_Em_Swc/StartBit:26/Length:2/J1939:YES *)
  S_Dr9_Opng : BOOL_T := (v := FALSE);  (* S_Dr9_Opng/StartBit:32/Length:2/J1939:YES *)
  S_Dr9_Clng : BOOL_T := (v := FALSE);  (* S_Dr9_Clng/StartBit:34/Length:2/J1939:YES *)
  S_Dr9_Op : BOOL_T := (v := FALSE);  (* S_Dr9_Op/StartBit:36/Length:2/J1939:YES *)
  S_Dr9_Cl : BOOL_T := (v := FALSE);  (* S_Dr9_Cl/StartBit:38/Length:2/J1939:YES *)
  S_Dr9_Obs : BOOL_T := (v := FALSE);  (* S_Dr9_Obs/StartBit:40/Length:2/J1939:YES *)
  S_Dr9_Em_Swc : BOOL_T := (v := FALSE);  (* S_Dr9_Em_Swc/StartBit:42/Length:2/J1939:YES *)
  X_Fus_0_D1 : BYTE_T := (v := FALSE);  (* ****************************************** MESSAGE: Sigorta_Kontrol_1 ID: 260 ****************************************** X_Fus_0_D1/StartBit:0/Length:8/J1939:NO *)
  X_Fus_0_D2 : BYTE_T := (v := FALSE);  (* X_Fus_0_D2/StartBit:8/Length:8/J1939:NO *)
  X_Fus_0_D3 : BYTE_T := (v := FALSE);  (* X_Fus_0_D3/StartBit:16/Length:8/J1939:NO *)
  X_Fus_0_D4 : BYTE_T := (v := FALSE);  (* X_Fus_0_D4/StartBit:24/Length:8/J1939:NO *)
  X_Fus_0_D5 : BYTE_T := (v := FALSE);  (* X_Fus_0_D5/StartBit:32/Length:8/J1939:NO *)
  X_Fus_0_D6 : BYTE_T := (v := FALSE);  (* X_Fus_0_D6/StartBit:40/Length:8/J1939:NO *)
  X_Fus_0_D7 : BYTE_T := (v := FALSE);  (* X_Fus_0_D7/StartBit:48/Length:8/J1939:NO *)
  X_Fus_0_D8 : BYTE_T := (v := FALSE);  (* X_Fus_0_D8/StartBit:56/Length:8/J1939:NO *)
  X_Fus_1_D1 : BYTE_T := (v := FALSE);  (* ****************************************** MESSAGE: Sigorta_Kontrol_2 ID: 261 ****************************************** X_Fus_1_D1/StartBit:0/Length:8/J1939:NO *)
  X_Fus_1_D2 : BYTE_T := (v := FALSE);  (* X_Fus_1_D2/StartBit:8/Length:8/J1939:NO *)
  X_Fus_1_D3 : BYTE_T := (v := FALSE);  (* X_Fus_1_D3/StartBit:16/Length:8/J1939:NO *)
  X_Fus_1_D4 : BYTE_T := (v := FALSE);  (* X_Fus_1_D4/StartBit:24/Length:8/J1939:NO *)
  X_Fus_1_D5 : BYTE_T := (v := FALSE);  (* X_Fus_1_D5/StartBit:32/Length:8/J1939:NO *)
  X_Fus_1_D6 : BYTE_T := (v := FALSE);  (* X_Fus_1_D6/StartBit:40/Length:8/J1939:NO *)
  X_Fus_1_D7 : BYTE_T := (v := FALSE);  (* X_Fus_1_D7/StartBit:48/Length:8/J1939:NO *)
  X_Fus_1_D8 : BYTE_T := (v := FALSE);  (* X_Fus_1_D8/StartBit:56/Length:8/J1939:NO *)
  X_Fus_2_D1 : BYTE_T := (v := FALSE);  (* ****************************************** MESSAGE: Sigorta_Kontrol_3 ID: 262 ****************************************** X_Fus_2_D1/StartBit:0/Length:8/J1939:NO *)
  X_Fus_2_D2 : BYTE_T := (v := FALSE);  (* X_Fus_2_D2/StartBit:8/Length:8/J1939:NO *)
  X_Fus_2_D3 : BYTE_T := (v := FALSE);  (* X_Fus_2_D3/StartBit:16/Length:8/J1939:NO *)
  X_Fus_2_D4 : BYTE_T := (v := FALSE);  (* X_Fus_2_D4/StartBit:24/Length:8/J1939:NO *)
  X_Fus_2_D5 : BYTE_T := (v := FALSE);  (* X_Fus_2_D5/StartBit:32/Length:8/J1939:NO *)
  X_Fus_2_D6 : BYTE_T := (v := FALSE);  (* X_Fus_2_D6/StartBit:40/Length:8/J1939:NO *)
  X_Fus_2_D7 : BYTE_T := (v := FALSE);  (* X_Fus_2_D7/StartBit:48/Length:8/J1939:NO *)
  X_Fus_2_D8 : BYTE_T := (v := FALSE);  (* X_Fus_2_D8/StartBit:56/Length:8/J1939:NO *)
  C_Param_Set : BOOL_T := (v := FALSE);  (* ****************************************** MESSAGE: DWP_Parameter ID: 263 ****************************************** C_Param_Set/StartBit:0/Length:2/J1939:YES *)
  P_Set_Tm_Dr_Cl_Rls : REAL_T := (v := FALSE);  (* P_Set_Tm_Dr_Cl_Rls/StartBit:8/Length:8/J1939:YES *)
  P_Set_Tm_Rout_Pnl_ShtDn : REAL_T := (v := FALSE);  (* P_Set_Tm_Vld_ShtDn/StartBit:16/Length:8/J1939:YES *)
  P_Set_Tm_Lgt_Dr_ShtDn : REAL_T := (v := FALSE);  (* P_Set_Tm_Lgt_Dr_ShtDn/StartBit:24/Length:8/J1939:YES *)
  X_Fus_3_D1 : BYTE_T := (v := FALSE);  (* ****************************************** MESSAGE: Sigorta_Kontrol_4 ID: 264 ****************************************** X_Fus_3_D1/StartBit:0/Length:8/J1939:NO *)
  X_Fus_3_D2 : BYTE_T := (v := FALSE);  (* X_Fus_3_D2/StartBit:8/Length:8/J1939:NO *)
  X_Fus_3_D3 : BYTE_T := (v := FALSE);  (* X_Fus_3_D3/StartBit:16/Length:8/J1939:NO *)
  X_Fus_3_D4 : BYTE_T := (v := FALSE);  (* X_Fus_3_D4/StartBit:24/Length:8/J1939:NO *)
  X_Fus_3_D5 : BYTE_T := (v := FALSE);  (* X_Fus_3_D5/StartBit:32/Length:8/J1939:NO *)
  X_Fus_3_D6 : BYTE_T := (v := FALSE);  (* X_Fus_3_D6/StartBit:40/Length:8/J1939:NO *)
  X_Fus_3_D7 : BYTE_T := (v := FALSE);  (* X_Fus_3_D7/StartBit:48/Length:8/J1939:NO *)
  X_Fus_3_D8 : BYTE_T := (v := FALSE);  (* X_Fus_3_D8/StartBit:56/Length:8/J1939:NO *)
  X_Sw_Ver_Mjr_DWP : REAL_T := (v := FALSE);  (* ****************************************** MESSAGE: Arac_Bilgisi_2 ID: 2E1 ****************************************** X_Sw_Ver_Mjr_DWP/StartBit:0/Length:8/J1939:YES *)
  X_Sw_Ver_Mnr_DWP : REAL_T := (v := FALSE);  (* X_Sw_Ver_Mnr_DWP/StartBit:8/Length:8/J1939:YES *)
  X_Sw_Ver_Tst_DWP : REAL_T := (v := FALSE);  (* X_Sw_Ver_Tst_DWP/StartBit:16/Length:8/J1939:YES *)
  X_Sw_Ver_Mjr_VCU : REAL_T := (v := FALSE);  (* X_Sw_Ver_Mjr_VCU/StartBit:24/Length:8/J1939:YES *)
  X_Sw_Ver_Mnr_VCU : REAL_T := (v := FALSE);  (* X_Sw_Ver_Mnr_VCU/StartBit:32/Length:8/J1939:YES *)
  X_Sw_Ver_Tst_VCU : REAL_T := (v := FALSE);  (* X_Sw_Ver_Tst_VCU/StartBit:40/Length:8/J1939:YES *)
  X_Sw_Ver_Mjr_ATS : REAL_T := (v := FALSE);  (* X_Sw_Ver_Mjr_ATS/StartBit:48/Length:8/J1939:YES *)
  X_Sw_Ver_Mnr_ATS : REAL_T := (v := FALSE);  (* X_Sw_Ver_Mnr_ATS/StartBit:54/Length:8/J1939:YES *)
  N_Diag_Lf : USINT_T := (v := FALSE);  (* ****************************************** MESSAGE: Diag_Temel_Durum ID: 300 ****************************************** N_Diag_Lf/StartBit:0/Length:8/J1939:YES *)
  C_Set_Odo_Btn : BOOL_T := (v := FALSE);  (* C_Set_Odo_Btn/StartBit:9/Length:1/J1939:YES *)
  S_Tst_Pg_Act : BOOL_T := (v := FALSE);  (* S_Tst_Pg_Act/StartBit:10/Length:2/J1939:YES *)
  S_Para_Pg_Act : BOOL_T := (v := FALSE);  (* S_Para_Pg_Act/StartBit:12/Length:2/J1939:YES *)
  S_HV_On_Btn : BOOL_T := (v := FALSE);  (* S_HV_On_Btn/StartBit:14/Length:1/J1939:NO *)
  S_HV_Off_Btn : BOOL_T := (v := FALSE);  (* S_HV_Off_Btn/StartBit:15/Length:1/J1939:NO *)
  S_Tm_Btn : BOOL_T := (v := FALSE);  (* S_Tm_Btn/StartBit:16/Length:1/J1939:NO *)
  S_Eep_Rst : BOOL_T := (v := FALSE);  (* S_Eep_Rst/StartBit:17/Length:1/J1939:NO *)
  C_Par_Rx : BOOL_T := (v := FALSE);  (* C_Par_Rx/StartBit:19/Length:1/J1939:NO *)
  C_Par_Wr : BOOL_T := (v := FALSE);  (* C_Par_Wr/StartBit:20/Length:1/J1939:NO *)
  C_Clr_EH : BOOL_T := (v := FALSE);  (* C_Clr_EH/StartBit:21/Length:1/J1939:NO *)
  S_Sw_Ver_Incomp : BOOL_T := (v := FALSE);  (* S_Sw_Ver_Incomp/StartBit:22/Length:1/J1939:NO *)
  W_Rd_Par_ID : REAL_T := (v := FALSE);  (* W_Rd_Par_ID/StartBit:24/Length:8/J1939:YES *)
  W_Odo : REAL_T := (v := FALSE);  (* W_Odo/StartBit:32/Length:32/J1939:YES *)
  X_Minute : REAL_T := (v := FALSE);  (* ****************************************** MESSAGE: Diag_RTC ID: 301 ****************************************** X_Minute/StartBit:0/Length:8/J1939:YES *)
  X_Hour : REAL_T := (v := FALSE);  (* X_Hour/StartBit:8/Length:8/J1939:YES *)
  X_Day : REAL_T := (v := FALSE);  (* X_Day/StartBit:16/Length:8/J1939:YES *)
  X_Month : REAL_T := (v := FALSE);  (* X_Month/StartBit:24/Length:8/J1939:YES *)
  X_Year : REAL_T := (v := FALSE);  (* X_Year/StartBit:32/Length:8/J1939:YES *)
  C_Rst_Tm_HVAC_On : BOOL_T := (v := FALSE);  (* ****************************************** MESSAGE: Diag_Op_Rst ID: 303 ****************************************** C_Rst_Tm_HVAC_On/StartBit:0/Length:1/J1939:NO *)
  C_Rst_Drv_Op_Cnt : BOOL_T := (v := FALSE);  (* C_Rst_Drv_Op_Cnt/StartBit:1/Length:1/J1939:NO *)
  C_Rst_Pass1_Op_Cnt : BOOL_T := (v := FALSE);  (* C_Rst_Pass1_Op_Cnt/StartBit:2/Length:1/J1939:NO *)
  C_Rst_Pass2_Op_Cnt : BOOL_T := (v := FALSE);  (* C_Rst_Pass2_Op_Cnt/StartBit:3/Length:1/J1939:NO *)
  C_Rst_Dr1_Cycle : BOOL_T := (v := FALSE);  (* C_Rst_Dr1_Cycle/StartBit:4/Length:1/J1939:NO *)
  C_Rst_Dr2_Cycle : BOOL_T := (v := FALSE);  (* C_Rst_Dr2_Cycle/StartBit:5/Length:1/J1939:NO *)
  C_Rst_Dr3_Cycle : BOOL_T := (v := FALSE);  (* C_Rst_Dr3_Cycle/StartBit:6/Length:1/J1939:NO *)
  C_Rst_Dr4_Cycle : BOOL_T := (v := FALSE);  (* C_Rst_Dr4_Cycle/StartBit:7/Length:1/J1939:NO *)
  S_Tst_HV_On : BOOL_T := (v := FALSE);  (* ****************************************** MESSAGE: ECU_Dijital_Cikis_Test ID: 310 ****************************************** S_Tst_HV_On/StartBit:34/Length:1/J1939:NO *)
  S_Tst_TCU_CAN_Sp : BOOL_T := (v := FALSE);  (* S_Tst_TCU_CAN_Sp/StartBit:37/Length:1/J1939:NO *)
  S_Tst_TCU_HV_On : BOOL_T := (v := FALSE);  (* S_Tst_TCU_HV_On/StartBit:38/Length:1/J1939:NO *)
  S_Tst_Air_Cmp_On : BOOL_T := (v := FALSE);  (* S_Tst_Air_Cmp_On/StartBit:39/Length:1/J1939:NO *)
  S_BMS_Wkup_Btn : BOOL_T := (v := FALSE);  (* S_BMS_Wkup_Btn/StartBit:40/Length:1/J1939:NO *)
  S_Mot_Fan_Ct_Btn : BOOL_T := (v := FALSE);  (* S_Mot_Fan_Ct_Btn/StartBit:41/Length:1/J1939:NO *)
  C_Flr_Heat_1_Ct : BOOL_T := (v := FALSE);  (* ****************************************** MESSAGE: Basamak_Isitici_Durumlari ID: 412 ****************************************** C_Flr_Heat_1_Ct/StartBit:0/Length:1/J1939:NO *)
  C_Flr_Heat_2_Ct : BOOL_T := (v := FALSE);  (* C_Flr_Heat_2_Ct/StartBit:1/Length:1/J1939:NO *)
  C_Flr_Heat_3_Ct : BOOL_T := (v := FALSE);  (* C_Flr_Heat_3_Ct/StartBit:2/Length:1/J1939:NO *)
  C_Flr_Heat_4_Ct : BOOL_T := (v := FALSE);  (* C_Flr_Heat_4_Ct/StartBit:3/Length:1/J1939:NO *)
  C_Flr_Heat_5_Ct : BOOL_T := (v := FALSE);  (* C_Flr_Heat_5_Ct/StartBit:4/Length:1/J1939:NO *)
  C_Flr_Heat_6_Ct : BOOL_T := (v := FALSE);  (* C_Flr_Heat_6_Ct/StartBit:5/Length:1/J1939:NO *)
  S_Flr_Heat_1 : BOOL_T := (v := FALSE);  (* S_Flr_Heat_1/StartBit:8/Length:1/J1939:NO *)
  S_Flr_Heat_2 : BOOL_T := (v := FALSE);  (* S_Flr_Heat_2/StartBit:9/Length:1/J1939:NO *)
  S_Flr_Heat_3 : BOOL_T := (v := FALSE);  (* S_Flr_Heat_3/StartBit:10/Length:1/J1939:NO *)
  S_Flr_Heat_4 : BOOL_T := (v := FALSE);  (* S_Flr_Heat_4/StartBit:11/Length:1/J1939:NO *)
  S_Flr_Heat_5 : BOOL_T := (v := FALSE);  (* S_Flr_Heat_5/StartBit:12/Length:1/J1939:NO *)
  S_Flr_Heat_6 : BOOL_T := (v := FALSE);  (* S_Flr_Heat_6/StartBit:13/Length:1/J1939:NO *)
  S_Flr_Heat_1_Fan_Actv : BOOL_T := (v := FALSE);  (* S_Flr_Heat_1_Fan_Actv/StartBit:16/Length:1/J1939:NO *)
  S_Flr_Heat_2_Fan_Actv : BOOL_T := (v := FALSE);  (* S_Flr_Heat_2_Fan_Actv/StartBit:17/Length:1/J1939:NO *)
  S_Flr_Heat_3_Fan_Actv : BOOL_T := (v := FALSE);  (* S_Flr_Heat_3_Fan_Actv/StartBit:18/Length:1/J1939:NO *)
  S_Flr_Heat_4_Fan_Actv : BOOL_T := (v := FALSE);  (* S_Flr_Heat_4_Fan_Actv/StartBit:19/Length:1/J1939:NO *)
  S_Flr_Heat_5_Fan_Actv : BOOL_T := (v := FALSE);  (* S_Flr_Heat_5_Fan_Actv/StartBit:20/Length:1/J1939:NO *)
  S_Flr_Heat_6_Fan_Actv : BOOL_T := (v := FALSE);  (* S_Flr_Heat_6_Fan_Actv/StartBit:21/Length:1/J1939:NO *)
  S_Flr_Heat_1_Fus_Blw : BOOL_T := (v := FALSE);  (* S_Flr_Heat_1_Fus_Blw/StartBit:24/Length:1/J1939:NO *)
  S_Flr_Heat_2_Fus_Blw : BOOL_T := (v := FALSE);  (* S_Flr_Heat_2_Fus_Blw/StartBit:25/Length:1/J1939:NO *)
  S_Flr_Heat_3_Fus_Blw : BOOL_T := (v := FALSE);  (* S_Flr_Heat_3_Fus_Blw/StartBit:26/Length:1/J1939:NO *)
  S_Flr_Heat_4_Fus_Blw : BOOL_T := (v := FALSE);  (* S_Flr_Heat_4_Fus_Blw/StartBit:27/Length:1/J1939:NO *)
  S_Flr_Heat_5_Fus_Blw : BOOL_T := (v := FALSE);  (* S_Flr_Heat_5_Fus_Blw/StartBit:28/Length:1/J1939:NO *)
  S_Flr_Heat_6_Fus_Blw : BOOL_T := (v := FALSE);  (* S_Flr_Heat_6_Fus_Blw/StartBit:29/Length:1/J1939:NO *)
  S_ER_Flr_Heat_1_Thstat : BOOL_T := (v := FALSE);  (* S_ER_Flr_Heat_1_Thstat/StartBit:32/Length:1/J1939:NO *)
  S_ER_Flr_Heat_2_Thstat : BOOL_T := (v := FALSE);  (* S_ER_Flr_Heat_2_Thstat/StartBit:33/Length:1/J1939:NO *)
  S_ER_Flr_Heat_3_Thstat : BOOL_T := (v := FALSE);  (* S_ER_Flr_Heat_3_Thstat/StartBit:34/Length:1/J1939:NO *)
  S_ER_Flr_Heat_4_Thstat : BOOL_T := (v := FALSE);  (* S_ER_Flr_Heat_4_Thstat/StartBit:35/Length:1/J1939:NO *)
  S_ER_Flr_Heat_5_Thstat : BOOL_T := (v := FALSE);  (* S_ER_Flr_Heat_5_Thstat/StartBit:36/Length:1/J1939:NO *)
  S_ER_Flr_Heat_6_Thstat : BOOL_T := (v := FALSE);  (* S_ER_Flr_Heat_6_Thstat/StartBit:37/Length:1/J1939:NO *)
  X_T_Flr_1 : REAL_T := (v := FALSE);  (* X_T_Flr_1/StartBit:40/Length:8/J1939:YES *)
  X_T_Flr_2 : REAL_T := (v := FALSE);  (* X_T_Flr_2/StartBit:48/Length:8/J1939:YES *)
  W_T_Flr : REAL_T := (v := FALSE);  (* W_T_Flr/StartBit:56/Length:8/J1939:YES *)
  S_TmOut_Haberlesme_Durumlari_0X200 : BOOL;  (* TIMEOUT SIGNALS Signal timeout status. Timeout parameter for signal :500ms *)
  S_TmOut_Direksiyon_Pompasi_Analog_0X210 : BOOL;  (* Signal timeout status. Timeout parameter for signal :500ms *)
  S_TmOut_Direksiyon_Pompasi_Durum_0X211 : BOOL;  (* Signal timeout status. Timeout parameter for signal :500ms *)
  S_TmOut_Arac_Durumlari_0X220 : BOOL;  (* Signal timeout status. Timeout parameter for signal :500ms *)
  S_TmOut_Fren_balata_durumlari_0X221 : BOOL;  (* Signal timeout status. Timeout parameter for signal :500ms *)
  S_TmOut_Fren_Basinclari_0X222 : BOOL;  (* Signal timeout status. Timeout parameter for signal :500ms *)
  S_TmOut_Lastik_Basinclari_1_0X223 : BOOL;  (* Signal timeout status. Timeout parameter for signal :500ms *)
  S_TmOut_Lastik_Basinclari_2_0X224 : BOOL;  (* Signal timeout status. Timeout parameter for signal :500ms *)
  S_TmOut_Arac_Bilgilendirme_0X225 : BOOL;  (* Signal timeout status. Timeout parameter for signal :500ms *)
  S_TmOut_Arac_Kritik_Uyarilari_0X226 : BOOL;  (* Signal timeout status. Timeout parameter for signal :500ms *)
  S_TmOut_Kapi_Hatalari_1_0X230 : BOOL;  (* Signal timeout status. Timeout parameter for signal :500ms *)
  S_TmOut_Kapi_Hatalari_2_0X231 : BOOL;  (* Signal timeout status. Timeout parameter for signal :500ms *)
  S_TmOut_Kapi_Hatalari_3_0X232 : BOOL;  (* Signal timeout status. Timeout parameter for signal :500ms *)
  S_TmOut_Kapi_Hatalari_4_0X233 : BOOL;  (* Signal timeout status. Timeout parameter for signal :500ms *)
  S_TmOut_Kapi_Hatalari_5_0X234 : BOOL;  (* Signal timeout status. Timeout parameter for signal :500ms *)
  S_TmOut_Kapi_Durum_1_0X235 : BOOL;  (* Signal timeout status. Timeout parameter for signal :500ms *)
  S_TmOut_Kapi_Durum_2_0X237 : BOOL;  (* Signal timeout status. Timeout parameter for signal :500ms *)
  S_TmOut_Kapi_Durum_3_0X238 : BOOL;  (* Signal timeout status. Timeout parameter for signal :500ms *)
  S_TmOut_Sigorta_Kontrol_1_0X260 : BOOL;  (* Signal timeout status. Timeout parameter for signal :500ms *)
  S_TmOut_Sigorta_Kontrol_2_0X261 : BOOL;  (* Signal timeout status. Timeout parameter for signal :500ms *)
  S_TmOut_Sigorta_Kontrol_3_0X262 : BOOL;  (* Signal timeout status. Timeout parameter for signal :500ms *)
  S_TmOut_Parametre_1_0X263 : BOOL;  (* Signal timeout status. Timeout parameter for signal :500ms *)
  S_TmOut_Sigorta_Kontrol_4_0X264 : BOOL;  (* Signal timeout status. Timeout parameter for signal :500ms *)
  S_TmOut_Diag_Temel_Durum_0X300 : BOOL;  (* Signal timeout status. Timeout parameter for signal :500ms *)
  S_TmOut_Diag_RTC_0X301 : BOOL;  (* Signal timeout status. Timeout parameter for signal :500ms *)
  S_TmOut_Diag_Parameter_0X302 : BOOL;  (* Signal timeout status. Timeout parameter for signal :500ms *)
  S_TmOut_Diag_Op_Rst_0X303 : BOOL;  (* Signal timeout status. Timeout parameter for signal :500ms *)
  S_TmOut_ECU_Dijital_Cikis_Test_0X310 : BOOL;  (* Signal timeout status. Timeout parameter for signal :500ms *)
  S_TmOut_Arac_Bilgi_2_0X2E1 : BOOL;  (* Signal timeout status. Timeout parameter for signal :500ms *)
  S_TmOut_Basamak_Isitici_Durumlari_0X412 : BOOL;  (* Signal timeout status. Timeout parameter for signal :5000ms *)
  S_Com_Flt : BOOL;  (* All of the timeout states are TRUE, no communication with unit *)
  S_Com_Distrb : BOOL;  (* One of the messages is not receiving from that unit, communication disturbed with unit *)
  S_CAN_Init : BOOL;  (* CAN Initilizer variable *)
END_STRUCT;
END_TYPE

TYPE DATAGRAM40_T : STRUCT
  ID0_LS : BYTE;
  ID0_HS : BYTE;
  ID0_Byte_0 : BYTE;
  ID0_Byte_1 : BYTE;
  ID0_Byte_2 : BYTE;
  ID0_Byte_3 : BYTE;
  ID0_Byte_4 : BYTE;
  ID0_Byte_5 : BYTE;
  ID0_Byte_6 : BYTE;
  ID0_Byte_7 : BYTE;
  ID1_LS : BYTE;
  ID1_HS : BYTE;
  ID1_Byte_0 : BYTE;
  ID1_Byte_1 : BYTE;
  ID1_Byte_2 : BYTE;
  ID1_Byte_3 : BYTE;
  ID1_Byte_4 : BYTE;
  ID1_Byte_5 : BYTE;
  ID1_Byte_6 : BYTE;
  ID1_Byte_7 : BYTE;
  ID2_LS : BYTE;
  ID2_HS : BYTE;
  ID2_Byte_0 : BYTE;
  ID2_Byte_1 : BYTE;
  ID2_Byte_2 : BYTE;
  ID2_Byte_3 : BYTE;
  ID2_Byte_4 : BYTE;
  ID2_Byte_5 : BYTE;
  ID2_Byte_6 : BYTE;
  ID2_Byte_7 : BYTE;
  ID3_LS : BYTE;
  ID3_HS : BYTE;
  ID3_Byte_0 : BYTE;
  ID3_Byte_1 : BYTE;
  ID3_Byte_2 : BYTE;
  ID3_Byte_3 : BYTE;
  ID3_Byte_4 : BYTE;
  ID3_Byte_5 : BYTE;
  ID3_Byte_6 : BYTE;
  ID3_Byte_7 : BYTE;
END_STRUCT;
END_TYPE

TYPE Eeprom_T : STRUCT
  P_Tm_Lf_Sign_TmOut_Dly : TIME := TIME#1s0ms;  (* The time paramter to wait set timeout on communication with a device *)
END_STRUCT;
END_TYPE

TYPE MSG_ETH_T : STRUCT
  X_Byte_0 : BYTE;
  X_Byte_1 : BYTE;
  X_Byte_2 : BYTE;
  X_Byte_3 : BYTE;
  X_Byte_4 : BYTE;
  X_Byte_5 : BYTE;
  X_Byte_6 : BYTE;
  X_Byte_7 : BYTE;
END_STRUCT;
END_TYPE

TYPE XTime_T : STRUCT
  X_Seconds : BYTE;
  X_Minutes : BYTE;
  X_Hours : BYTE;
  X_Days : BYTE;
  X_Months : BYTE;
  X_Years : BYTE;
END_STRUCT;
END_TYPE

TYPE IOVD_T : STRUCT
  X_Param_Arr : Param_T;
  S_ER_Com_VCU : BOOL_T := (v := FALSE);  (* ****************************************** MESSAGE: ECU_Haberlesme ID: 400 ****************************************** S_ER_Com_VCU/StartBit:0/Length:2/J1939:YES *)
  S_ER_Com_TCU : BOOL_T := (v := FALSE);  (* S_ER_Com_TCU/StartBit:2/Length:2/J1939:YES *)
  S_ER_Com_ESS : BOOL_T := (v := FALSE);  (* S_ER_Com_ESS/StartBit:4/Length:2/J1939:YES *)
  S_ER_Com_HVAC : BOOL_T := (v := FALSE);  (* S_ER_Com_HVAC/StartBit:6/Length:2/J1939:YES *)
  S_ER_Com_EBS : BOOL_T := (v := FALSE);  (* S_ER_Com_EBS/StartBit:12/Length:2/J1939:YES *)
  S_ER_Com_PCAN : BOOL_T := (v := FALSE);  (* S_ER_Com_PCAN/StartBit:14/Length:2/J1939:YES *)
  S_ER_Com_Pnt : BOOL_T := (v := FALSE);  (* S_ER_Com_Pnt/StartBit:16/Length:2/J1939:YES *)
  S_ER_Com_Acc_Pdl : BOOL_T := (v := FALSE);  (* S_ER_Com_Acc_Pdl/StartBit:18/Length:2/J1939:YES *)
  S_ER_Com_Str_Ang_Snsr : BOOL_T := (v := FALSE);  (* S_ER_Com_Str_Ang_Snsr/StartBit:20/Length:2/J1939:YES *)
  S_PDU_Cvr_Op : BOOL_T := (v := FALSE);  (* S_PDU_Cvr_Op/StartBit:22/Length:2/J1939:YES *)
  S_ER_HVAC_Amb : BOOL_T := (v := FALSE);  (* S_ER_HVAC_Amb/StartBit:24/Length:1/J1939:NO *)
  S_ER_HVAC_Red : BOOL_T := (v := FALSE);  (* S_ER_HVAC_Red/StartBit:25/Length:1/J1939:NO *)
  S_ER_Iso_Amb : BOOL_T := (v := FALSE);  (* S_ER_Iso_Amb/StartBit:26/Length:1/J1939:NO *)
  S_ER_Iso_Red : BOOL_T := (v := FALSE);  (* S_ER_Iso_Red/StartBit:27/Length:1/J1939:NO *)
  S_ER_Amb : BOOL_T := (v := FALSE);  (* S_ER_Amb/StartBit:28/Length:1/J1939:NO *)
  S_ER_Red : BOOL_T := (v := FALSE);  (* S_ER_Red/StartBit:29/Length:1/J1939:NO *)
  S_Rdy_Dep : BOOL_T := (v := FALSE);  (* S_Rdy_Dep/StartBit:30/Length:1/J1939:NO *)
  S_Pwr_Red : BOOL_T := (v := FALSE);  (* S_Pwr_Red/StartBit:31/Length:1/J1939:NO *)
  S_ER_BCU_Amb : BOOL_T := (v := FALSE);  (* S_ER_BCU_Amb/StartBit:32/Length:1/J1939:NO *)
  S_ER_BCU_Red : BOOL_T := (v := FALSE);  (* S_ER_BCU_Red/StartBit:33/Length:1/J1939:NO *)
  S_ER_Temp_Red : BOOL_T := (v := FALSE);  (* S_ER_Temp_Red/StartBit:34/Length:1/J1939:NO *)
  S_ER_Temp_Amb : BOOL_T := (v := FALSE);  (* S_ER_Temp_Amb/StartBit:35/Length:1/J1939:NO *)
  S_ER_HV_Amb : BOOL_T := (v := FALSE);  (* S_ER_HV_Amb/StartBit:36/Length:1/J1939:NO *)
  S_ER_HV_Red : BOOL_T := (v := FALSE);  (* S_ER_HV_Red/StartBit:37/Length:1/J1939:NO *)
  S_ER_Pnt_Amb : BOOL_T := (v := FALSE);  (* S_ER_Pnt_Amb/StartBit:38/Length:1/J1939:NO *)
  S_ER_Pnt_Red : BOOL_T := (v := FALSE);  (* S_ER_Pnt_Red/StartBit:39/Length:1/J1939:NO *)
  S_Mot_Temp_Hi : BOOL_T := (v := FALSE);  (* S_Mot_Temp_Hi/StartBit:45/Length:1/J1939:NO *)
  S_Mot_Temp_Too_Hi : BOOL_T := (v := FALSE);  (* S_Mot_Temp_Too_Hi/StartBit:46/Length:1/J1939:NO *)
  S_ER_BCCU : BOOL_T := (v := FALSE);  (* S_ER_BCCU/StartBit:47/Length:1/J1939:NO *)
  S_Ln_Vo_Lo : BOOL_T := (v := FALSE);  (* S_Ln_Vo_Lo/StartBit:48/Length:1/J1939:NO *)
  S_Ln_Vo_Hi : BOOL_T := (v := FALSE);  (* S_Ln_Vo_Too_Lo/StartBit:49/Length:1/J1939:NO *)
  S_ER_Mot_Cnv_Amb : BOOL_T := (v := FALSE);  (* S_ER_Mot_Cnv_Amb/StartBit:50/Length:1/J1939:NO *)
  S_ER_Mot_Cnv_Red : BOOL_T := (v := FALSE);  (* S_ER_Mot_Cnv_Red/StartBit:51/Length:1/J1939:NO *)
  S_ER_Icy_Road_Amb : BOOL_T := (v := FALSE);  (* S_ER_Icy_Road_Amb/StartBit:52/Length:1/J1939:NO *)
  S_ER_Str_Pmp_Temp_Hi : BOOL_T := (v := FALSE);  (* S_ER_Str_Pmp_Temp_Hi/StartBit:53/Length:1/J1939:NO *)
  S_ER_Aux_AC_Amb : BOOL_T := (v := FALSE);  (* S_ER_Aux_AC_Amb/StartBit:54/Length:1/J1939:NO *)
  S_ER_Aux_AC_Red : BOOL_T := (v := FALSE);  (* S_ER_Aux_AC_Red/StartBit:55/Length:1/J1939:NO *)
  Z_Vh_Mode : BYTE_T := (v := FALSE);  (* Vehicle_mode_bitmask/StartBit:56/Length:8/J1939:YES *)
  X_DDS_No_1 : REAL_T := (v := FALSE);  (* ****************************************** MESSAGE: DDS ID: 401 ****************************************** X_DDS_No_1/StartBit:0/Length:16/J1939:YES *)
  X_DDS_No_2 : REAL_T := (v := FALSE);  (* X_DDS_No_2/StartBit:16/Length:16/J1939:YES *)
  X_DDS_No_3 : REAL_T := (v := FALSE);  (* X_DDS_No_3/StartBit:32/Length:16/J1939:YES *)
  X_DDS_No_4 : REAL_T := (v := FALSE);  (* X_DDS_No_4/StartBit:48/Length:16/J1939:YES *)
  X_DDS_No_5 : REAL_T := (v := FALSE);  (* ****************************************** MESSAGE: DDS_2 ID: 402 ****************************************** X_DDS_No_5/StartBit:0/Length:16/J1939:YES *)
  X_Tot_Pg_No : REAL_T := (v := FALSE);  (* X_Tot_Pg_No/StartBit:16/Length:8/J1939:YES *)
  X_Cur_Pg_No : REAL_T := (v := FALSE);  (* X_Cur_Pg_No/StartBit:24/Length:8/J1939:YES *)
  S_ER_Susp_Amb : BOOL;  (* ****************************************** MESSAGE: ECU Parametre ID: 403 ****************************************** S_ER_Susp_Amb/StartBit:0/Length:1/J1939:YES *)
  S_ER_Susp_Red : BOOL;  (* S_ER_Susp_Red/StartBit:1/Length:1/J1939:YES *)
  S_ER_Lo_Pr_Amb : BOOL;  (* S_ER_Lo_Pr_Amb/StartBit:2/Length:1/J1939:YES *)
  S_ER_Lo_Pr_Red : BOOL;  (* S_ER_Lo_Pr_Red/StartBit:3/Length:1/J1939:YES *)
  S_ER_Ret : BOOL;  (* S_ER_Ret/StartBit:4/Length:1/J1939:YES *)
  P_X_Tm_Dr_Cl_Rls : REAL_T := (v := FALSE);  (* P_X_Tm_Dr_Cl_Rls/StartBit:8/Length:8/J1939:YES *)
  P_X_Tm_Vld_ShtDn : REAL_T := (v := FALSE);  (* P_X_Tm_Vld_ShtDn/StartBit:16/Length:8/J1939:YES *)
  P_X_Tm_Lgt_Dr_ShtDn : REAL_T := (v := FALSE);  (* P_X_Tm_Lgt_Dr_ShtDn/StartBit:24/Length:8/J1939:YES *)
  S_HVAC_Sp : BOOL_T := (v := FALSE);  (* ****************************************** MESSAGE: HVAC_Durum ID: 410 ****************************************** S_HVAC_Sp/StartBit:0/Length:2/J1939:YES *)
  S_HVAC_Mn_Swc : BOOL_T := (v := FALSE);  (* S_HVAC_Mn_Swc/StartBit:2/Length:2/J1939:YES *)
  S_HVAC_Otp_Do : BOOL_T := (v := FALSE);  (* S_HVAC_Otp_Do/StartBit:4/Length:2/J1939:YES *)
  C_Dmst_On : BOOL_T := (v := FALSE);  (* C_Dmst_On/StartBit:6/Length:2/J1939:YES *)
  S_BTMS_En : BOOL_T := (v := FALSE);  (* S_BTMS_En/StartBit:8/Length:2/J1939:YES *)
  S_Elec_Heat_1_En : BOOL_T := (v := FALSE);  (* S_Elec_Heat_1_En/StartBit:10/Length:2/J1939:YES *)
  S_Elec_Heat_2_En : BOOL_T := (v := FALSE);  (* S_Elec_Heat_2_En/StartBit:12/Length:2/J1939:YES *)
  S_HVAC_Inver_En : BOOL_T := (v := FALSE);  (* S_HVAC_Inver_En/StartBit:14/Length:2/J1939:YES *)
  S_HVAC_1_En : BOOL_T := (v := FALSE);  (* S_HVAC_1_En/StartBit:16/Length:2/J1939:YES *)
  S_HVAC_2_En : BOOL_T := (v := FALSE);  (* S_HVAC_2_En/StartBit:18/Length:2/J1939:YES *)
  S_HVAC_Drv_En : BOOL_T := (v := FALSE);  (* S_HVAC_Drv_En/StartBit:20/Length:2/J1939:YES *)
  S_BTMS_Actv : BOOL_T := (v := FALSE);  (* S_BTMS_Actv/StartBit:24/Length:2/J1939:YES *)
  Z_BTMS_Mode : BYTE_T := (v := FALSE);  (* Z_BTMS_Mode/StartBit:26/Length:2/J1939:YES *)
  Z_BTMS_Req_Mode : BYTE_T := (v := FALSE);  (* Z_BTMS_Req_Mode/StartBit:28/Length:2/J1939:YES *)
  S_Elec_Heat_1_On : BOOL_T := (v := FALSE);  (* S_Elec_Heat_1_On/StartBit:30/Length:2/J1939:YES *)
  S_Elec_Heat_2_On : BOOL_T := (v := FALSE);  (* S_Elec_Heat_2_On/StartBit:32/Length:2/J1939:YES *)
  S_HVAC_Inver_On : BOOL_T := (v := FALSE);  (* S_HVAC_Inver_On/StartBit:34/Length:2/J1939:YES *)
  S_Elec_Heat_Tm_On : BOOL_T := (v := FALSE);  (* S_Elec_Heat_Tm_On/StartBit:36/Length:2/J1939:YES *)
  Z_HVAC_1_Mode : BYTE_T := (v := FALSE);  (* Z_HVAC_1_Mode/StartBit:40/Length:4/J1939:YES *)
  Z_HVAC_2_Mode : BYTE_T := (v := FALSE);  (* Z_HVAC_2_Mode/StartBit:44/Length:4/J1939:YES *)
  Z_HVAC_Drv_Mode : BYTE_T := (v := FALSE);  (* Z_HVAC_Drv_Mode/StartBit:48/Length:4/J1939:YES *)
  Z_ER_HVAC : BYTE_T := (v := FALSE);  (* Z_ER_HVAC/StartBit:52/Length:4/J1939:YES *)
  X_Spd_HVAC_Fan : REAL_T := (v := FALSE);  (* X_Spd_HVAC_Fan/StartBit:56/Length:8/J1939:YES *)
  X_T_Drv : REAL_T := (v := FALSE);  (* ****************************************** MESSAGE: HVAC_Sicaklik ID: 411 ****************************************** X_T_Drv/StartBit:0/Length:8/J1939:YES *)
  W_T_Drv : REAL_T := (v := FALSE);  (* W_T_Drv/StartBit:8/Length:8/J1939:YES *)
  X_T_Insd_1 : REAL_T := (v := FALSE);  (* X_T_Insd_1/StartBit:16/Length:8/J1939:YES *)
  X_T_Insd_2 : REAL_T := (v := FALSE);  (* X_T_Insd_2/StartBit:24/Length:8/J1939:YES *)
  W_T_HVAC_Psng : REAL_T := (v := FALSE);  (* W_T_HVAC_Psng/StartBit:32/Length:8/J1939:YES *)
  X_T_Amb : REAL_T := (v := FALSE);  (* X_T_Amb/StartBit:40/Length:8/J1939:YES *)
  X_T_Clt_Wtr : REAL_T := (v := FALSE);  (* X_T_Clt_Wtr/StartBit:48/Length:8/J1939:YES *)
  X_P_HVAC_Inver : REAL_T := (v := FALSE);  (* ****************************************** MESSAGE: HVAC_Analog ID: 413 ****************************************** X_P_HVAC_Inver/StartBit:0/Length:16/J1939:YES *)
  X_P_Elec_Heat : REAL_T := (v := FALSE);  (* X_P_Elec_Heat/StartBit:16/Length:16/J1939:YES *)
  X_I_In_HVAC_Inver : REAL_T := (v := FALSE);  (* X_I_In_HVAC_Inver/StartBit:32/Length:16/J1939:YES *)
  X_I_In_Elec_Heat : REAL_T := (v := FALSE);  (* X_I_In_Elec_Heat/StartBit:48/Length:16/J1939:YES *)
  C_Defrs_Plus_Ct : BOOL_T := (v := FALSE);  (* ****************************************** MESSAGE: Klima_Kontaktor_Kontrol ID: 414 ****************************************** C_Defrs_Plus_Ct/StartBit:0/Length:1/J1939:NO *)
  C_Defrs_Minus_Ct : BOOL_T := (v := FALSE);  (* C_Defrs_Minus_Ct/StartBit:1/Length:1/J1939:NO *)
  C_Prheat_Plus_Ct : BOOL_T := (v := FALSE);  (* C_Prheat_Plus_Ct/StartBit:2/Length:1/J1939:NO *)
  C_Prheat_Minus_Ct : BOOL_T := (v := FALSE);  (* C_Prheat_Minus_Ct/StartBit:3/Length:1/J1939:NO *)
  C_HVAC_Plus_Ct : BOOL_T := (v := FALSE);  (* C_HVAC_Plus_Ct/StartBit:4/Length:1/J1939:NO *)
  C_HVAC_Minus_Ct : BOOL_T := (v := FALSE);  (* C_HVAC_Minus_Ct/StartBit:5/Length:1/J1939:NO *)
  S_Defrs_Plus_Ct_Deactv : BOOL_T := (v := FALSE);  (* S_Defrs_Plus_Ct_Deactv/StartBit:6/Length:1/J1939:NO *)
  S_Defrs_Minus_Ct_Deactv : BOOL_T := (v := FALSE);  (* S_Defrs_Minus_Ct_Deactv/StartBit:7/Length:1/J1939:NO *)
  S_Prheat_Plus_Ct_Deactv : BOOL_T := (v := FALSE);  (* S_Prheat_Plus_Ct_Deactv/StartBit:8/Length:1/J1939:NO *)
  S_Prheat_Minus_Ct_Deactv : BOOL_T := (v := FALSE);  (* S_Prheat_Minus_Ct_Deactv/StartBit:9/Length:1/J1939:NO *)
  S_HVAC_Plus_Ct_Deactv : BOOL_T := (v := FALSE);  (* S_HVAC_Plus_Ct_Deactv/StartBit:10/Length:1/J1939:NO *)
  S_HVAC_Minus_Ct_Deactv : BOOL_T := (v := FALSE);  (* S_HVAC_Minus_Ct_Deactv/StartBit:11/Length:1/J1939:NO *)
  Z_Btms_Stat : BYTE_T := (v := FALSE);  (* Z_Btms_Stat/StartBit:12/Length:4/J1939:NO *)
  Z_HvacDrv_Stat : BYTE_T := (v := FALSE);  (* Z_HvacDrv_Stat/StartBit:16/Length:8/J1939:NO *)
  Z_HvacPass1_Stat : BYTE_T := (v := FALSE);  (* Z_HvacPass1_Stat/StartBit:24/Length:8/J1939:NO *)
  Z_HvacPass2_Stat : BYTE_T := (v := FALSE);  (* Z_HvacPass2_Stat/StartBit:32/Length:8/J1939:NO *)
  Z_Elec_Heaters_Stat : BYTE_T := (v := FALSE);  (* Z_Elec_Heaters_Stat/StartBit:40/Length:8/J1939:NO *)
  Z_Flr_Heaters_Stat_1 : BYTE_T := (v := FALSE);  (* Z_Flr_Heaters_Stat_1/StartBit:48/Length:8/J1939:NO *)
  Z_Flr_Heaters_Stat_2 : BYTE_T := (v := FALSE);  (* Z_Flr_Heaters_Stat_2/StartBit:56/Length:8/J1939:NO *)
  P_X_T_Max_Bat_BTMS_Heat : REAL_T := (v := FALSE);  (* ****************************************** MESSAGE: HVAC_Parameters_1 ID: 415 ****************************************** P_X_T_Max_Bat_BTMS_Heat/StartBit:0/Length:8/J1939:YES *)
  P_X_T_Max_Bat_BTMS_Cool : REAL_T := (v := FALSE);  (* P_X_T_Max_Bat_BTMS_Cool/StartBit:8/Length:8/J1939:YES *)
  P_X_T_Max_Wtr_BTMS_Heat : REAL_T := (v := FALSE);  (* P_X_T_Max_Wtr_BTMS_Heat/StartBit:16/Length:8/J1939:YES *)
  P_X_T_Max_Wtr_BTMS_Cool : REAL_T := (v := FALSE);  (* P_X_T_Max_Wtr_BTMS_Cool/StartBit:24/Length:8/J1939:YES *)
  P_X_T_Flr_Heat_Lim : REAL_T := (v := FALSE);  (* P_X_T_Flr_Heat_Lim/StartBit:32/Length:8/J1939:YES *)
  X_T_BTMS_Wtr_Snsr_1 : REAL_T := (v := FALSE);  (* ****************************************** MESSAGE: HVAC_Water_Temperature ID: 416 ****************************************** X_T_BTMS_Wtr_Snsr_1/StartBit:0/Length:8/J1939:YES *)
  X_T_BTMS_Wtr_Snsr_2 : REAL_T := (v := FALSE);  (* X_T_BTMS_Wtr_Snsr_2/StartBit:8/Length:8/J1939:YES *)
  S_ESS_Mn_Ct : BOOL_T := (v := FALSE);  (* ****************************************** MESSAGE: ESS_Durum ID: 430 ****************************************** S_ESS_Mn_Ct/StartBit:0/Length:2/J1939:YES *)
  S_Insu_Ok : BOOL_T := (v := FALSE);  (* S_Insu_Ok/StartBit:4/Length:2/J1939:YES *)
  S_BMS_Sp : BOOL_T := (v := FALSE);  (* S_BMS_Sp/StartBit:6/Length:2/J1939:YES *)
  S_Bat_Mode : BOOL_T := (v := FALSE);  (* S_Bat_Mode/StartBit:8/Length:2/J1939:YES *)
  S_Ops_Mode : BOOL_T := (v := FALSE);  (* S_Ops_Mode/StartBit:10/Length:2/J1939:YES *)
  C_Tr_Mode : BOOL_T := (v := FALSE);  (* C_Tr_Mode/StartBit:12/Length:2/J1939:YES *)
  S_Pwr_Distr : BOOL_T := (v := FALSE);  (* S_Pwr_Distr/StartBit:16/Length:2/J1939:YES *)
  S_Ext_Sp_Req : BOOL_T := (v := FALSE);  (* S_Ext_Sp_Req/StartBit:24/Length:2/J1939:YES *)
  X_Vh_Mode_Req : BYTE_T := (v := FALSE);  (* S_Vh_Mode_Req/StartBit:26/Length:2/J1939:YES *)
  Z_MBMS_Mode : BYTE_T := (v := FALSE);  (* Z_MBMS_Mode/StartBit:32/Length:8/J1939:YES *)
  Z_Bat_Ops : BYTE_T := (v := FALSE);  (* Z_Bat_Ops/StartBit:40/Length:4/J1939:YES *)
  C_BMS_Wkup : BOOL_T := (v := FALSE);  (* C_BMS_Wkup/StartBit:44/Length:2/J1939:YES *)
  Z_Bat_Mode : BYTE_T := (v := FALSE);  (* Z_Bat_Mode/StartBit:48/Length:8/J1939:YES *)
  Z_ESS_Stat : BYTE_T := (v := FALSE);  (* Z_ESS_Stat/StartBit:56/Length:8/J1939:YES *)
  X_U_Bat_1 : REAL_T := (v := FALSE);  (* ****************************************** MESSAGE: ESS_Paket_Voltaji ID: 431 ****************************************** X_U_Bat_1/StartBit:0/Length:16/J1939:YES *)
  X_U_Bat_2 : REAL_T := (v := FALSE);  (* X_U_Bat_2/StartBit:16/Length:16/J1939:YES *)
  X_U_Bat_3 : REAL_T := (v := FALSE);  (* X_U_Bat_3/StartBit:32/Length:16/J1939:YES *)
  X_U_Bat_4 : REAL_T := (v := FALSE);  (* X_U_Bat_4/StartBit:48/Length:16/J1939:YES *)
  X_I_Bat_1 : REAL_T := (v := FALSE);  (* ****************************************** MESSAGE: ESS_Paket_Akim ID: 432 ****************************************** X_I_Bat_1/StartBit:0/Length:16/J1939:YES *)
  X_I_Bat_2 : REAL_T := (v := FALSE);  (* X_I_Bat_2/StartBit:16/Length:16/J1939:YES *)
  X_I_Bat_3 : REAL_T := (v := FALSE);  (* X_I_Bat_3/StartBit:32/Length:16/J1939:YES *)
  X_I_Bat_4 : REAL_T := (v := FALSE);  (* X_I_Bat_4/StartBit:48/Length:16/J1939:YES *)
  X_U_Max_Bat_1 : REAL_T := (v := FALSE);  (* ****************************************** MESSAGE: ESS_Maksimum_Hucre_Voltaji ID: 433 ****************************************** X_U_Max_Cell_1/StartBit:0/Length:16/J1939:YES *)
  X_U_Max_Bat_2 : REAL_T := (v := FALSE);  (* X_U_Max_Cell_2/StartBit:16/Length:16/J1939:YES *)
  X_U_Max_Bat_3 : REAL_T := (v := FALSE);  (* X_U_Max_Cell_3/StartBit:32/Length:16/J1939:YES *)
  X_U_Max_Bat_4 : REAL_T := (v := FALSE);  (* X_U_Max_Cell_4/StartBit:48/Length:16/J1939:YES *)
  X_U_Min_Bat_1 : REAL_T := (v := FALSE);  (* ****************************************** MESSAGE: ESS_Minimum_Hucre_Voltaji ID: 434 ****************************************** X_U_Min_Cell_1/StartBit:0/Length:16/J1939:YES *)
  X_U_Min_Bat_2 : REAL_T := (v := FALSE);  (* X_U_Min_Cell_2/StartBit:16/Length:16/J1939:YES *)
  X_U_Min_Bat_3 : REAL_T := (v := FALSE);  (* X_U_Min_Cell_3/StartBit:32/Length:16/J1939:YES *)
  X_U_Min_Bat_4 : REAL_T := (v := FALSE);  (* X_U_Min_Cell_4/StartBit:48/Length:16/J1939:YES *)
  X_U_Avg_Cell_1 : REAL_T := (v := FALSE);  (* ****************************************** MESSAGE: ESS_Ortalama_Hucre_Voltaji ID: 435 ****************************************** X_U_Avg_Cell_1/StartBit:0/Length:16/J1939:YES *)
  X_U_Avg_Cell_2 : REAL_T := (v := FALSE);  (* X_U_Avg_Cell_2/StartBit:16/Length:16/J1939:YES *)
  X_U_Avg_Cell_3 : REAL_T := (v := FALSE);  (* X_U_Avg_Cell_3/StartBit:32/Length:16/J1939:YES *)
  X_U_Avg_Cell_4 : REAL_T := (v := FALSE);  (* X_U_Avg_Cell_4/StartBit:48/Length:16/J1939:YES *)
  X_T_Max_Bat_1 : REAL_T := (v := FALSE);  (* ****************************************** MESSAGE: ESS_Sicaklik ID: 436 ****************************************** X_T_Max_Cell_1/StartBit:0/Length:8/J1939:YES *)
  X_T_Max_Bat_2 : REAL_T := (v := FALSE);  (* X_T_Max_Cell_2/StartBit:8/Length:8/J1939:YES *)
  X_T_Max_Bat_3 : REAL_T := (v := FALSE);  (* X_T_Max_Cell_3/StartBit:16/Length:8/J1939:YES *)
  X_T_Min_Bat_1 : REAL_T := (v := FALSE);  (* X_T_Min_Cell_1/StartBit:32/Length:8/J1939:YES *)
  X_T_Min_Bat_2 : REAL_T := (v := FALSE);  (* X_T_Min_Cell_2/StartBit:40/Length:8/J1939:YES *)
  X_T_Min_Bat_3 : REAL_T := (v := FALSE);  (* X_T_Min_Cell_3/StartBit:48/Length:8/J1939:YES *)
  X_T_Avg_Bat_1 : REAL_T := (v := FALSE);  (* X_T_Avg_Bat_1/StartBit:56/Length:8/J1939:YES *)
  X_I_Max_Chrg : REAL_T := (v := FALSE);  (* ****************************************** MESSAGE: ESS_Analog ID: 437 ****************************************** X_I_Max_Chrg/StartBit:16/Length:16/J1939:YES *)
  X_I_Max_Dischrg : REAL_T := (v := FALSE);  (* X_I_Max_Dischrg/StartBit:32/Length:16/J1939:YES *)
  X_U_Tot_Bat : REAL_T := (v := FALSE);  (* X_U_Tot_Bat/StartBit:48/Length:16/J1939:YES *)
  W_T_Clt : REAL_T := (v := FALSE);  (* ****************************************** MESSAGE: ESS_Sogutma_Suyu ID: 438 ****************************************** W_T_Clt/StartBit:0/Length:8/J1939:YES *)
  X_T_Clt : REAL_T := (v := FALSE);  (* X_T_Clt/StartBit:8/Length:8/J1939:YES *)
  C_Ign_Hv_On : BOOL_T := (v := FALSE);  (* ****************************************** MESSAGE: HV_Durum ID: 450 ****************************************** C_Ign_Hv_On/StartBit:0/Length:2/J1939:YES *)
  C_Pnt_Hv_On : BOOL_T := (v := FALSE);  (* C_Pnt_Hv_On/StartBit:6/Length:2/J1939:YES *)
  C_Bat_Lo_Hv_On : BOOL_T := (v := FALSE);  (* C_Bat_Lo_Hv_On/StartBit:8/Length:2/J1939:YES *)
  C_Tm_Hv_On : BOOL_T := (v := FALSE);  (* C_Tm_Hv_On/StartBit:10/Length:2/J1939:YES *)
  C_Diag_Hv_On : BOOL_T := (v := FALSE);  (* C_Diag_Hv_On/StartBit:12/Length:2/J1939:YES *)
  C_Ign_Hv_Off : BOOL_T := (v := FALSE);  (* C_Ign_Hv_Off/StartBit:16/Length:2/J1939:YES *)
  C_Pnt_Hv_Off : BOOL_T := (v := FALSE);  (* C_Pnt_Hv_Off/StartBit:22/Length:2/J1939:YES *)
  C_Bat_Lo_Hv_Off : BOOL_T := (v := FALSE);  (* C_Bat_Lo_Hv_Off/StartBit:24/Length:2/J1939:YES *)
  C_Tm_Hv_Off : BOOL_T := (v := FALSE);  (* C_Tm_Hv_Off/StartBit:26/Length:2/J1939:YES *)
  C_Diag_Hv_Off : BOOL_T := (v := FALSE);  (* C_Diag_Hv_Off/StartBit:28/Length:2/J1939:YES *)
  C_Hv_On : BOOL_T := (v := FALSE);  (* C_Hv_On/StartBit:32/Length:2/J1939:YES *)
  C_Hv_Off : BOOL_T := (v := FALSE);  (* C_Hv_Off/StartBit:34/Length:2/J1939:YES *)
  S_Hv_On_Prc : BOOL_T := (v := FALSE);  (* S_Hv_On_Prc/StartBit:36/Length:2/J1939:YES *)
  S_Hv_Off_Prc : BOOL_T := (v := FALSE);  (* S_Hv_Off_Prc/StartBit:38/Length:2/J1939:YES *)
  S_Em_Stop : BOOL_T := (v := FALSE);  (* S_Em_Stop/StartBit:40/Length:2/J1939:YES *)
  S_Hv_On_En : BOOL_T := (v := FALSE);  (* S_Hv_On_En/StartBit:42/Length:2/J1939:YES *)
  S_Hv_Off_En : BOOL_T := (v := FALSE);  (* S_Hv_Off_En/StartBit:44/Length:2/J1939:YES *)
  C_Mn_Ct_On : BOOL_T := (v := FALSE);  (* C_Mn_Ct_On/StartBit:46/Length:2/J1939:YES *)
  S_Mn_Ct : BOOL_T := (v := FALSE);  (* S_Mn_Ct/StartBit:48/Length:2/J1939:YES *)
  C_Prechrg_Ct_On : BOOL_T := (v := FALSE);  (* C_Prechrg_Ct_On/StartBit:50/Length:2/J1939:YES *)
  S_Prechrg_Ct : BOOL_T := (v := FALSE);  (* S_Prechrg_Ct/StartBit:52/Length:2/J1939:YES *)
  S_ER_HV : BOOL_T := (v := FALSE);  (* S_ER_HV/StartBit:54/Length:2/J1939:YES *)
  S_ER_Mn_Ct : BOOL_T := (v := FALSE);  (* S_ER_Mn_Ct/StartBit:56/Length:2/J1939:YES *)
  S_ER_Prechrg_Ct : BOOL_T := (v := FALSE);  (* S_ER_Prechrg_Ct/StartBit:58/Length:2/J1939:YES *)
  S_Hv_On : BOOL_T := (v := FALSE);  (* S_Hv_On/StartBit:60/Length:2/J1939:YES *)
  S_HV_HVAC_En : BOOL_T := (v := FALSE);  (* S_HV_HVAC_En/StartBit:62/Length:2/J1939:YES *)
  S_Mn_Ct_Req : BOOL_T := (v := FALSE);  (* ****************************************** MESSAGE: TCU_Trolleybus_Durum ID: 460 ****************************************** S_Mn_Ct_Req/StartBit:0/Length:2/J1939:YES *)
  S_Sys_On : BOOL_T := (v := FALSE);  (* S_Sys_On/StartBit:2/Length:2/J1939:YES *)
  S_Mot_Cnv_On_Req : BOOL_T := (v := FALSE);  (* S_Mot_Cnv_On_Req/StartBit:4/Length:2/J1939:YES *)
  S_Mot_Cnv_On : BOOL_T := (v := FALSE);  (* S_Mot_Cnv_On/StartBit:6/Length:2/J1939:YES *)
  S_24V_Bat_Cnv_On_Req : BOOL_T := (v := FALSE);  (* S_24V_Bat_Cnv_On_Req/StartBit:8/Length:2/J1939:YES *)
  S_24V_Sp_On : BOOL_T := (v := FALSE);  (* S_24V_Sp_On/StartBit:10/Length:2/J1939:YES *)
  S_Pnt_Chrg_Req : BOOL_T := (v := FALSE);  (* S_Pnt_Chrg_Req/StartBit:12/Length:2/J1939:YES *)
  S_Pnt_Chrg_Fdbk : BOOL_T := (v := FALSE);  (* S_Pnt_Chrg_Fdbk/StartBit:14/Length:2/J1939:YES *)
  Z_Drv_Dir_Req : BYTE_T := (v := FALSE);  (* Z_Drv_Dir_Req/StartBit:16/Length:2/J1939:YES *)
  Z_Drv_Dir : BYTE_T := (v := FALSE);  (* Z_Drv_Dir/StartBit:18/Length:2/J1939:YES *)
  S_Elec_Mode_Req : BOOL_T := (v := FALSE);  (* S_Elec_Mode_Req/StartBit:20/Length:2/J1939:YES *)
  S_Elec_Mode_Actv : BOOL_T := (v := FALSE);  (* S_Elec_Mode_Actv/StartBit:22/Length:2/J1939:YES *)
  S_Bat_Mode_Req : BOOL_T := (v := FALSE);  (* S_Bat_Mode_Req/StartBit:24/Length:2/J1939:YES *)
  S_Bat_Mode_Actv : BOOL_T := (v := FALSE);  (* S_Bat_Mode_Actv/StartBit:26/Length:2/J1939:YES *)
  S_Elec_Ret_En : BOOL_T := (v := FALSE);  (* S_Elec_Ret_En/StartBit:28/Length:2/J1939:YES *)
  S_Elec_Brk_En : BOOL_T := (v := FALSE);  (* S_Elec_Brk_En/StartBit:30/Length:2/J1939:YES *)
  S_Tintl : BOOL_T := (v := FALSE);  (* S_Tintl/StartBit:32/Length:2/J1939:YES *)
  S_Em_Deact : BOOL_T := (v := FALSE);  (* S_Em_Deact/StartBit:34/Length:2/J1939:YES *)
  S_Rs_Cosu_Req : BOOL_T := (v := FALSE);  (* S_Rs_Cosu_Req/StartBit:36/Length:2/J1939:YES *)
  S_TCU_Hlt_Brk_Req : BOOL_T := (v := FALSE);  (* S_TCU_Hlt_Brk_Req/StartBit:38/Length:2/J1939:YES *)
  S_Insu_Test_Mod_Actv : BOOL_T := (v := FALSE);  (* S_Insu_Test_Mod_Actv/StartBit:40/Length:2/J1939:YES *)
  S_Engy_Flw_Trol : BOOL_T := (v := FALSE);  (* S_Engy_Flw_Trol/StartBit:42/Length:2/J1939:YES *)
  S_Engy_Flw_Bat : BOOL_T := (v := FALSE);  (* S_Engy_Flw_Bat/StartBit:44/Length:2/J1939:YES *)
  S_Trol_Volt_Actv : BOOL_T := (v := FALSE);  (* S_Trol_Volt_Actv/StartBit:46/Length:2/J1939:YES *)
  C_Mot_Fan_Ct : BOOL_T := (v := FALSE);  (* C_Mot_Fan_Ct/StartBit:48/Length:2/J1939:YES *)
  S_Mot_Fan_Thrm_Ct : BOOL_T := (v := FALSE);  (* S_Mot_Fan_Thrm_Ct/StartBit:50/Length:2/J1939:YES *)
  S_ER_Elec_Brk_Amb : BOOL_T := (v := FALSE);  (* S_ER_Elec_Brk_Amb/StartBit:52/Length:2/J1939:YES *)
  S_ER_Elec_Brk_Red : BOOL_T := (v := FALSE);  (* S_ER_Elec_Brk_Red/StartBit:54/Length:2/J1939:YES *)
  Z_Mc_Stat : BYTE_T := (v := FALSE);  (* Z_Mc_Stat/StartBit:56/Length:2/J1939:YES *)
  X_Spd_Max_Fwd : REAL_T := (v := FALSE);  (* ****************************************** MESSAGE: TCU_Surus_Limit ID: 462 ****************************************** X_Spd_Max_Fwd/StartBit:0/Length:8/J1939:YES *)
  X_Spd_Max_Bwd : REAL_T := (v := FALSE);  (* X_Spd_Max_Bwd/StartBit:8/Length:8/J1939:YES *)
  X_Ang_Str : REAL_T := (v := FALSE);  (* X_Ang_Str/StartBit:16/Length:8/J1939:YES *)
  X_Pct_Brk_Pdl : REAL_T := (v := FALSE);  (* X_Pct_Brk_Pdl/StartBit:32/Length:8/J1939:YES *)
  X_Pct_Acc_Pdl : REAL_T := (v := FALSE);  (* X_Pct_Acc_Pdl/StartBit:40/Length:8/J1939:YES *)
  S_Hlt_Brk_Actv : BOOL_T := (v := FALSE);  (* S_Hlt_Brk_Actv/StartBit:48/Length:2/J1939:YES *)
  X_T_Mot : REAL_T := (v := FALSE);  (* ****************************************** MESSAGE: TCU_Analog ID: 463 ****************************************** X_T_Mot/StartBit:0/Length:8/J1939:YES *)
  X_T_Mot_Cnv : REAL_T := (v := FALSE);  (* X_T_Mot_Cnv/StartBit:8/Length:8/J1939:YES *)
  X_T_TCU_Box : REAL_T := (v := FALSE);  (* X_T_TCU_Box/StartBit:16/Length:8/J1939:YES *)
  X_P_ESS : REAL_T := (v := FALSE);  (* X_P_ESS/StartBit:32/Length:16/J1939:YES *)
  X_I_Out_ESS : REAL_T := (v := FALSE);  (* X_I_Out_ESS/StartBit:48/Length:16/J1939:YES *)
  X_I_Out_Mot_Cnv : REAL_T := (v := FALSE);  (* ****************************************** MESSAGE: TCU_Cikis_Akim_Guc ID: 464 ****************************************** X_I_Out_Mot_Cnv/StartBit:0/Length:16/J1939:YES *)
  X_I_Brk_Rsr : REAL_T := (v := FALSE);  (* X_I_Brk_Rsr/StartBit:16/Length:16/J1939:YES *)
  X_P_Mot_Cnv : REAL_T := (v := FALSE);  (* X_P_Mot_Cnv/StartBit:32/Length:16/J1939:YES *)
  X_P_Brk_Rsr : REAL_T := (v := FALSE);  (* X_P_Brk_Rsr/StartBit:48/Length:16/J1939:YES *)
  X_M_Act : REAL_T := (v := FALSE);  (* ****************************************** MESSAGE: TCU_Tork_Hiz ID: 465 ****************************************** X_M_Act/StartBit:0/Length:16/J1939:YES *)
  X_Spd_Act : REAL_T := (v := FALSE);  (* X_Spd_Act/StartBit:16/Length:16/J1939:YES *)
  X_Spd_Act_kmh : REAL_T := (v := FALSE);  (* X_Spd_Act_kmh/StartBit:32/Length:16/J1939:YES *)
  N_Tm_Trol_Md : UDINT_T := (v := FALSE);  (* ****************************************** MESSAGE: TCU_Calisma_Suresi ID: 466 ****************************************** N_Tm_Trol_Md/StartBit:0/Length:32/J1939:YES *)
  N_Tm_Bat_Md : UDINT_T := (v := FALSE);  (* N_Tm_Bat_Md/StartBit:32/Length:32/J1939:YES *)
  X_U_Inv_HV : REAL_T := (v := FALSE);  (* ****************************************** MESSAGE: TCU_Analog_2 ID: 467 ****************************************** X_U_Inv_HV/StartBit:0/Length:16/J1939:YES *)
  X_U_Cat_Ln : REAL_T := (v := FALSE);  (* X_U_Cat_Ln/StartBit:16/Length:16/J1939:YES *)
  S_Aux_AC_Cnv_Rdy : BOOL_T := (v := FALSE);  (* ****************************************** MESSAGE: Yardimci_Konvertor_Durum ID: 480 ****************************************** S_Aux_AC_Cnv_Rdy/StartBit:0/Length:2/J1939:YES *)
  C_Aux_AC_Cnv_On : BOOL_T := (v := FALSE);  (* C_Aux_AC_Cnv_On/StartBit:2/Length:2/J1939:YES *)
  S_Aux_AC_Cnv_On : BOOL_T := (v := FALSE);  (* S_Aux_AC_Cnv_On/StartBit:4/Length:2/J1939:YES *)
  S_Aux_DC_24V_Cnv_Rdy : BOOL_T := (v := FALSE);  (* S_Aux_DC_24V_Cnv_Rdy/StartBit:6/Length:2/J1939:YES *)
  C_Aux_DC_24V_Cnv_On : BOOL_T := (v := FALSE);  (* C_Aux_DC_24V_Cnv_On/StartBit:8/Length:2/J1939:YES *)
  S_Aux_DC_24V_Cnv_On : BOOL_T := (v := FALSE);  (* S_Aux_DC_24V_Cnv_On/StartBit:10/Length:2/J1939:YES *)
  C_Aux_DC_Cnv_On : BOOL_T := (v := FALSE);  (* C_Aux_DC_Cnv_On/StartBit:12/Length:2/J1939:YES *)
  S_Aux_DC_Cnv_On : BOOL_T := (v := FALSE);  (* S_Aux_DC_Cnv_On/StartBit:14/Length:2/J1939:YES *)
  C_Bat_Chrg_DC_Cnv_On : BOOL_T := (v := FALSE);  (* C_Bat_Chrg_DC_Cnv_On/StartBit:16/Length:2/J1939:YES *)
  S_Bat_Chrg_DC_Cnv_On : BOOL_T := (v := FALSE);  (* S_Bat_Chrg_DC_Cnv_On/StartBit:18/Length:2/J1939:YES *)
  C_Aux_DC_Ct_1_On : BOOL_T := (v := FALSE);  (* C_Aux_DC_Ct_1_On/StartBit:20/Length:2/J1939:YES *)
  C_Aux_DC_Ct_2_On : BOOL_T := (v := FALSE);  (* C_Aux_DC_Ct_2_On/StartBit:22/Length:2/J1939:YES *)
  C_Aux_DC_Ct_3_On : BOOL_T := (v := FALSE);  (* C_Aux_DC_Ct_3_On/StartBit:24/Length:2/J1939:YES *)
  S_Aux_DC_Ct_1_Actv : BOOL_T := (v := FALSE);  (* S_Aux_DC_Ct_1_Actv/StartBit:26/Length:2/J1939:YES *)
  S_Aux_DC_Ct_2_Actv : BOOL_T := (v := FALSE);  (* S_Aux_DC_Ct_2_Actv/StartBit:28/Length:2/J1939:YES *)
  S_Aux_DC_Ct_3_Actv : BOOL_T := (v := FALSE);  (* S_Aux_DC_Ct_3_Actv/StartBit:30/Length:2/J1939:YES *)
  Z_Bccu_Stat : BYTE_T := (v := FALSE);  (* Z_Bccu_Stat/StartBit:32/Length:8/J1939:YES *)
  Z_Tcu_Stat : BYTE_T := (v := FALSE);  (* Z_Tcu_Stat/StartBit:40/Length:8/J1939:YES *)
  Z_Apu_Stat : BYTE_T := (v := FALSE);  (* Z_Apu_Stat/StartBit:48/Length:8/J1939:YES *)
  X_I_Out_Aux_DC_Cnv : REAL_T := (v := FALSE);  (* ****************************************** MESSAGE: Yardimci_Konvertor_Akim ID: 481 ****************************************** X_I_Out_Aux_DC_Cnv/StartBit:0/Length:16/J1939:YES *)
  X_I_Out_Aux_AC_Cnv : REAL_T := (v := FALSE);  (* X_I_Out_Aux_AC_Cnv/StartBit:16/Length:16/J1939:YES *)
  X_I_Out_Aux_DC_24V_Cnv : REAL_T := (v := FALSE);  (* X_I_Out_Aux_DC_24V_Cnv/StartBit:32/Length:16/J1939:YES *)
  X_I_In_Aux_DC_24V_Cnv : REAL_T := (v := FALSE);  (* X_I_In_Aux_DC_24V_Cnv/StartBit:48/Length:16/J1939:YES *)
  X_U_Out_24V_Bat : REAL_T := (v := FALSE);  (* ****************************************** MESSAGE: Yardimci_Konvertor_Guc ID: 482 ****************************************** X_U_Out_24V_Bat/StartBit:0/Length:16/J1939:YES *)
  X_P_Out_Aux_DC_Cnv : REAL_T := (v := FALSE);  (* X_P_Out_Aux_DC_Cnv/StartBit:16/Length:16/J1939:YES *)
  X_P_Out_Aux_AC_Cnv : REAL_T := (v := FALSE);  (* X_P_Out_Aux_AC_Cnv/StartBit:32/Length:16/J1939:YES *)
  X_P_Out_Aux_DC_24V_Cnv : REAL_T := (v := FALSE);  (* X_P_Out_Aux_DC_24V_Cnv/StartBit:48/Length:16/J1939:YES *)
  X_P_Bat_Chrg_DC_Cnv : REAL_T := (V := FALSE);  (* ****************************************** MESSAGE: Batarya_Konvertor_Analog ID: 483 ****************************************** X_P_Bat_Chrg_DC_Cnv/StartBit:0/Length:16/J1939:YES *)
  X_I_Out_Aux_Bat_Chrg_DC_Cnv : REAL_T := (V := FALSE);  (* X_I_Out_Aux_Bat_Chrg_DC_Cnv/StartBit:16/Length:16/J1939:YES *)
  X_T_Aux_AC_Cnv : REAL_T := (v := FALSE);  (* ****************************************** MESSAGE: Yardimci_Konvertor_Sicaklik ID: 484 ****************************************** X_T_Aux_AC_Cnv/StartBit:0/Length:8/J1939:YES *)
  X_T_Aux_DC_24V_Cnv : REAL_T := (v := FALSE);  (* X_T_Aux_DC_24V_Cnv/StartBit:8/Length:8/J1939:YES *)
  X_T_Aux_DC_Cnv : REAL_T := (v := FALSE);  (* X_T_Aux_DC_Cnv/StartBit:16/Length:8/J1939:YES *)
  X_T_Bat_Chrg_DC_Cnv : REAL_T := (v := FALSE);  (* X_T_Bat_Chrg_DC_Cnv/StartBit:24/Length:8/J1939:YES *)
  Z_Insu_Dev : BYTE_T := (v := FALSE);  (* ****************************************** MESSAGE: Isolation_Status ID: 485 ****************************************** Z_Insu_Dev/StartBit:0/Length:5/J1939:YES *)
  S_ER_Insu_Dev_Not_Conn : BOOL_T := (v := FALSE);  (* S_ER_Insu_Dev_Not_Conn/StartBit:4/Length:1/J1939:YES *)
  Z_Man_Insu_Tst : BYTE_T := (v := FALSE);  (* Z_Man_Insu_Tst/StartBit:8/Length:8/J1939:YES *)
  Z_Semi_Aut_Insu_Tst : BYTE_T := (v := FALSE);  (* Z_Semi_Aut_Insu_Tst/StartBit:16/Length:8/J1939:YES *)
  S_Insu_Tst_Ok : BOOL_T := (v := FALSE);  (* S_Insu_Tst_Ok/StartBit:24/Length:1/J1939:YES *)
  S_Man_Insu_Meas_Actv : BOOL_T := (v := FALSE);  (* S_Man_Insu_Meas_Actv/StartBit:25/Length:2/J1939:YES *)
  S_Aut_Insu_Meas_Actv : BOOL_T := (v := FALSE);  (* S_Aut_Insu_Meas_Actv/StartBit:25/Length:2/J1939:YES *)
  S_Vh_Chrg_Perm : BOOL_T := (v := FALSE);  (* ****************************************** MESSAGE: Sarj_Durum ID: 4A0 ****************************************** S_Vh_Chrg_Perm/StartBit:0/Length:2/J1939:YES *)
  S_Vh_Insu_Meas : BOOL_T := (v := FALSE);  (* S_Vh_Insu_Meas/StartBit:2/Length:2/J1939:YES *)
  S_Vh_Mobil : BOOL_T := (v := FALSE);  (* S_Vh_Mobil/StartBit:4/Length:2/J1939:YES *)
  S_Chrg_Cmpl : BOOL_T := (v := FALSE);  (* S_Chrg_Cmpl/StartBit:8/Length:2/J1939:YES *)
  S_EV_Rdy : BOOL_T := (v := FALSE);  (* S_EV_Rdy/StartBit:10/Length:2/J1939:YES *)
  C_Chrg_Btn_Lft_Bwd_Led_Ctrl : BOOL_T := (v := FALSE);  (* C_Chrg_Btn_Lft_Bwd_Led_Ctrl/Startbit:12/Length:2/J1939:YES *)
  S_Pnt_Chrg_Mode_Sel : BOOL_T := (v := FALSE);  (* S_Pnt_Chrg_Mode_Sel/StartBit:16/Length:2/J1939:YES *)
  S_Pnt_Chrg_Mode : BOOL_T := (v := FALSE);  (* S_Pnt_Chrg_Mode/StartBit:18/Length:2/J1939:YES *)
  S_TCU_Pnt_Chrg_Ct : BOOL_T := (v := FALSE);  (* S_TCU_Pnt_Chrg_Ct/StartBit:20/Length:2/J1939:YES *)
  S_TCU_Chrg_Ct : BOOL_T := (v := FALSE);  (* S_TCU_Chrg_Ct/StartBit:22/Length:2/J1939:YES *)
  X_Tm_Seri_Hour : REAL_T := (v := FALSE);  (* ****************************************** MESSAGE: Sarj_Sureleri ID: 4A5 ****************************************** X_Tm_Seri_Hour/StartBit:0/Length:8/J1939:YES *)
  X_Tm_Seri_Minute : REAL_T := (v := FALSE);  (* X_Tm_Seri_Minute/StartBit:8/Length:8/J1939:YES *)
  X_Tm_Sp_Mode_Hour : REAL_T := (v := FALSE);  (* X_Tm_Sp_Mode_Hour/StartBit:32/Length:8/J1939:YES *)
  X_Tm_Sp_Mode_Minute : REAL_T := (v := FALSE);  (* X_Tm_Sp_Mode_Minute/StartBit:40/Length:8/J1939:YES *)
  X_Tm_Estm_Fn_Hour : REAL_T := (v := FALSE);  (* X_Tm_Estm_Fn_Hour/StartBit:48/Length:8/J1939:YES *)
  X_Tm_Estm_Fn_Minute : REAL_T := (v := FALSE);  (* X_Tm_Estm_Fn_Minute/StartBit:56/Length:8/J1939:YES *)
  Z_Ext_Chrg_Stat : BYTE_T := (v := FALSE);  (* ****************************************** MESSAGE: Sarj_Durum_3 ID: 4A6 ****************************************** Z_Ext_Chrg_Stat/StartBit:0/Length:8/J1939:YES *)
  Z_Pan_Chrg_Stat : BYTE_T := (v := FALSE);  (* Z_Pan_Chrg_Stat/StartBit:8/Length:8/J1939:YES *)
  Z_Pnt_Pos : BYTE_T := (v := FALSE);  (* Z_Pnt_Pos/StartBit:16/Length:8/J1939:YES *)
  X_I_Pnt_Chrg : REAL_T := (v := FALSE);  (* ****************************************** MESSAGE: Pantograph_Analog_4 ID: 4AF ****************************************** X_I_Pnt_Chrg/StartBit:0/Length:16/J1939:YES *)
  X_U_Pnt_Chrg : REAL_T := (v := FALSE);  (* X_U_Pnt_Chrg/StartBit:16/Length:16/J1939:YES *)
  X_P_Pnt_Chrg : REAL_T := (v := FALSE);  (* X_P_Pnt_Chrg/StartBit:32/Length:16/J1939:YES *)
  X_T_Pnt_Chrg : REAL_T := (v := FALSE);  (* X_T_Pnt_Chrg/StartBit:48/Length:16/J1939:YES *)
  X_I_Lft_AC_Chrg : REAL_T := (v := FALSE);  (* ****************************************** MESSAGE: Left_Charge_Analog_1 ID: 4B0 ****************************************** X_I_Lft_AC_Chrg/StartBit:0/Length:16/J1939:YES *)
  X_U_Lft_AC_Chrg : REAL_T := (v := FALSE);  (* X_U_Lft_AC_Chrg/StartBit:16/Length:16/J1939:YES *)
  X_Capcty_Lft_AC_Chrg : REAL_T := (v := FALSE);  (* X_Capcty_Lft_AC_Chrg/StartBit:32/Length:32/J1939:YES *)
  X_Distn_Bat_Drvn : REAL_T := (v := FALSE);  (* ****************************************** MESSAGE: Arac_Menzil ID: 4C0 ****************************************** X_Distn_Bat_Drvn/StartBit:0/Length:16/J1939:YES *)
  X_Distn_Rmn : REAL_T := (v := FALSE);  (* X_Distn_Rmn/StartBit:16/Length:16/J1939:YES *)
  X_Distn_Cat_Drvn : REAL_T := (v := FALSE);  (* X_Distn_Cat_Drvn/StartBit:32/Length:32/J1939:YES *)
  X_Om : REAL_T := (v := FALSE);  (* ****************************************** MESSAGE: Arac_Odometre ID: 4C1 ****************************************** X_Om/StartBit:0/Length:32/J1939:YES *)
  X_Spd_TCU : REAL_T := (v := FALSE);  (* ****************************************** MESSAGE: Arac_Genel_Istatistik ID: 4C2 ****************************************** X_Spd_TCU/StartBit:0/Length:8/J1939:YES *)
  X_Spd_EBS : REAL_T := (v := FALSE);  (* X_Spd_EBS/StartBit:8/Length:8/J1939:YES *)
  X_SOC : REAL_T := (v := FALSE);  (* X_SOC/StartBit:16/Length:8/J1939:YES *)
  X_SOH : REAL_T := (v := FALSE);  (* X_SOH/StartBit:24/Length:8/J1939:YES *)
  X_Accl : REAL_T := (v := FALSE);  (* X_Accl/StartBit:32/Length:16/J1939:YES *)
  X_Cosu_Avg : REAL_T := (v := FALSE);  (* X_Cosu_Avg/StartBit:48/Length:16/J1939:YES *)
  X_E_Tr : REAL_T := (v := FALSE);  (* ****************************************** MESSAGE: Arac_Surus_Enerji ID: 4C3 ****************************************** X_E_Tr/StartBit:0/Length:32/J1939:YES *)
  X_E_Regn : REAL_T := (v := FALSE);  (* X_E_Regn/StartBit:32/Length:32/J1939:YES *)
  X_E_Aux_DC : REAL_T := (v := FALSE);  (* ****************************************** MESSAGE: Arac_Tuketilen_Enerji_1 ID: 4C4 ****************************************** X_E_Aux_DC/StartBit:0/Length:32/J1939:YES *)
  X_E_Aux_DC_24V : REAL_T := (v := FALSE);  (* X_E_Aux_DC_24V/StartBit:32/Length:32/J1939:YES *)
  X_E_Aux_AC : REAL_T := (v := FALSE);  (* ****************************************** MESSAGE: Arac_Tuketilen_Enerji_2 ID: 4C5 ****************************************** X_E_Aux_AC/StartBit:0/Length:32/J1939:YES *)
  X_E_Cosu : REAL_T := (v := FALSE);  (* X_E_Cosu/StartBit:32/Length:32/J1939:YES *)
  X_Capcty_Act : REAL_T := (v := FALSE);  (* ****************************************** MESSAGE: Arac_Kapasite ID: 4C6 ****************************************** X_Capcty_Act/StartBit:0/Length:32/J1939:YES *)
  X_Capcty_Rmn : REAL_T := (v := FALSE);  (* X_Capcty_Rmn/StartBit:32/Length:32/J1939:YES *)
  X_Tm_Bat_Drvn : REAL_T := (v := FALSE);  (* ****************************************** MESSAGE: Arac_Sureler ID: 4C7 ****************************************** X_Tm_Bat_Drvn/StartBit:0/Length:16/J1939:YES *)
  X_Tm_Cat_Drvn : REAL_T := (v := FALSE);  (* X_Tm_Cat_Drvn/StartBit:16/Length:16/J1939:YES *)
  X_Tm_Wt : REAL_T := (v := FALSE);  (* X_Tm_Wt/StartBit:32/Length:16/J1939:YES *)
  X_Tm_HVAC_On : REAL_T := (v := FALSE);  (* X_Tm_HVAC_On/StartBit:48/Length:16/J1939:YES *)
  X_E_Tot_Cosu : REAL_T := (v := FALSE);  (* ****************************************** MESSAGE: Arac_Toplam_Tuketilen_Enerji ID: 4C8 ****************************************** X_E_Tot_Cosu/StartBit:0/Length:32/J1939:YES *)
  X_Avg_Cosu_Opp : REAL_T := (v := FALSE);  (* X_Avg_Cosu_Opp/StartBit:32/Length:16/J1939:YES *)
  X_Daily_Avg_Cosu : REAL_T := (v := FALSE);  (* ****************************************** MESSAGE: Arac_Genel_Istatistik_2 ID: 4C9 ****************************************** X_Daily_Avg_Cosu/StartBit:0/Length:16/J1939:YES *)
  X_Trp_Distn : REAL_T := (v := FALSE);  (* X_Trp_Distn/StartBit:16/Length:32/J1939:YES *)
  X_U_ECU_Sp : REAL_T := (v := FALSE);  (* X_U_ECU_Sp/StartBit:48/Length:16/J1939:YES *)
  N_Hvac_Drv_Op_Cnt : UDINT_T := (v := FALSE);  (* ****************************************** MESSAGE: Klima_Calisma_Sureleri_1 ID: 4CA ****************************************** N_Hvac_Drv_Op_Cnt/StartBit:0/Length:32/J1939:YES *)
  N_Hvac_Pass1_Op_Cnt : UDINT_T := (v := FALSE);  (* N_Hvac_Pass1_Op_Cnt/StartBit:32/Length:32/J1939:YES *)
  N_Hvac_Pass2_Op_Cnt : UDINT_T := (v := FALSE);  (* ****************************************** MESSAGE: Klima_Calisma_Sureleri_2 ID: 4CB ****************************************** N_Hvac_Pass2_Op_Cnt/StartBit:0/Length:32/J1939:YES *)
  N_Btms_Op_Cnt : UDINT_T := (v := FALSE);  (* N_Btms_Op_Cnt/StartBit:32/Length:32/J1939:YES *)
  N_Air_Cmp_Op_Cnt : UDINT_T := (v := FALSE);  (* ****************************************** MESSAGE: Sayicilar_1 ID: 4CC ****************************************** N_Air_Cmp_Op_Cnt/StartBit:0/Length:32/J1939:YES *)
  X_Opp_Dist_Bat : REAL_T := (v := FALSE);  (* X_Opp_Dist_Bat/StartBit:32/Length:16/J1939:NO *)
  X_E_Aux_Cons : REAL_T := (v := FALSE);  (* ****************************************** MESSAGE: Yardimci_Tuketici_Enerjileri ID: 4CD ****************************************** X_E_Aux_Cons/StartBit:0/Length:32/J1939:YES *)
  X_E_Aux_Hvac_Cons : REAL_T := (v := FALSE);  (* X_E_Aux_Hvac_Cons/StartBit:32/Length:32/J1939:YES *)
  N_Dr1_Cycle : REAL_T := (v := FALSE);  (* ****************************************** MESSAGE: Kapi_Sayicilari_1 ID: 4CD ****************************************** N_Dr1_Cycle/StartBit:0/Length:32/J1939:NO *)
  N_Dr2_Cycle : REAL_T := (v := FALSE);  (* N_Dr2_Cycle/StartBit:32/Length:32/J1939:NO *)
  N_Dr3_Cycle : REAL_T := (v := FALSE);  (* ****************************************** MESSAGE: Kapi_Sayicilari_2 ID: 4CE ****************************************** N_Dr3_Cycle/StartBit:0/Length:32/J1939:NO *)
  N_Dr4_Cycle : REAL_T := (v := FALSE);  (* N_Dr4_Cycle/StartBit:32/Length:32/J1939:NO *)
  X_E_Chrg_Pan : REAL_T := (v := FALSE);  (* ****************************************** MESSAGE: Sarj_Enerjisi ID: 4CF ****************************************** X_E_Chrg_Pan/StartBit:32/Length:32/J1939:NO *)
  X_E_Chrg_Onbrd : REAL_T := (v := FALSE);  (* X_E_Chrg_Onbrd/StartBit:0/Length:32/J1939:NO *)
  X_Vh_No : REAL_T := (v := FALSE);  (* ****************************************** MESSAGE: Arac_Bilgi_1 ID: 4E0 ****************************************** X_Vh_No/StartBit:0/Length:16/J1939:YES *)
  X_Sw_Ver_Mjr_ECU : REAL_T := (v := FALSE);  (* X_Sw_Ver_Mjr_ECU/StartBit:16/Length:8/J1939:YES *)
  X_Sw_Ver_Mnr_ECU : REAL_T := (v := FALSE);  (* X_Sw_Ver_Mnr_ECU/StartBit:24/Length:8/J1939:YES *)
  X_Sw_Ver_Tst_ECU : REAL_T := (v := FALSE);  (* X_Sw_Ver_Tst_ECU/StartBit:32/Length:8/J1939:YES *)
  X_Sw_Ver_Mjr_TCU : REAL_T := (v := FALSE);  (* X_Sw_Ver_Mjr_TCU/StartBit:24/Length:8/J1939:YES *)
  X_Sw_Ver_Mnr_TCU : REAL_T := (v := FALSE);  (* X_Sw_Ver_Mnr_TCU/StartBit:32/Length:8/J1939:YES *)
  X_Sw_Ver_Tst_TCU : REAL_T := (v := FALSE);  (* X_Sw_Ver_Tst_TCU/StartBit:40/Length:8/J1939:YES *)
  C_Air_Cmp_On : BOOL_T := (v := FALSE);  (* ****************************************** MESSAGE: Hava_Kompresoru_Durum ID: 4F0 ****************************************** C_Air_Cmp_On/StartBit:0/Length:2/J1939:YES *)
  S_Air_Cmp_On : BOOL_T := (v := FALSE);  (* S_Air_Cmp_On/StartBit:2/Length:2/J1939:YES *)
  S_ER_Air_Cmp : BOOL_T := (v := FALSE);  (* S_ER_Air_Cmp/StartBit:4/Length:2/J1939:YES *)
  S_ER_Hi_Temp_Air_Cmp : BOOL_T := (v := FALSE);  (* S_ER_Hi_Temp_Air_Cmp/StartBit:6/Length:2/J1939:YES *)
  S_ER_Psb_Air_Lek : BOOL_T := (v := FALSE);  (* S_ER_Psb_Air_Lek/StartBit:8/Length:2/J1939:YES *)
  X_Tot_TypA_Evnt : WORD_T := (v := FALSE);  (* ****************************************** MESSAGE: Olay_Durum ID: 500 ****************************************** X_Tot_TypA_Evnt/StartBit:0/Length:16/J1939:NO *)
  X_Tot_TypB_Evnt : WORD_T := (v := FALSE);  (* X_Tot_TypB_Evnt/StartBit:16/Length:16/J1939:NO *)
  N_ECU_Lf : USINT_T := (v := FALSE);  (* ****************************************** MESSAGE: Temel_Durum ID: 99 ****************************************** N_ECU_Lf/StartBit:0/Length:8/J1939:YES *)
  S_Sw_Up_Avl : BOOL_T := (v := FALSE);  (* S_Sw_Up_Avl/StartBit:8/Length:2/J1939:YES *)
  S_EH_Rd_Avl : BOOL_T := (v := FALSE);  (* S_EH_Rd_Avl/StartBit:10/Length:2/J1939:YES *)
  S_Tst_Avl : BOOL_T := (v := FALSE);  (* S_Tst_Avl/StartBit:12/Length:2/J1939:YES *)
  S_Para_Up_Avl : BOOL_T := (v := FALSE);  (* S_Para_Up_Avl/StartBit:14/Length:2/J1939:YES *)
  C_ECU_Rst : BOOL_T := (v := FALSE);  (* C_ECU_Rst/StartBit:16/Length:2/J1939:YES *)
  S_Brk_Tst_Mode : BOOL_T := (v := FALSE);  (* S_Brk_Tst_Mode/StartBit:18/Length:2/J1939:YES *)
  Z_Vh_Typ : BYTE_T := (v := FALSE);  (* Z_Vh_Typ/StartBit:32/Length:8/J1939:YES *)
  X_Prj_No : REAL_T := (v := FALSE);  (* X_Prj_No/StartBit:48/Length:16/J1939:YES *)
  S_SentOk_Parametre_0X101 : BOOL;  (* Message sent SIGNALS Message sent status provided by LIB500 *)
  S_SentOk_ECU_Haberlesme_0X400 : BOOL;  (* Message sent status provided by LIB500 *)
  C_En_ECU_Haberlesme_0X400 : BOOL;  (* Message enable bit for message ID 16#400 *)
  S_SentOk_DDS_0X401 : BOOL;  (* Message sent status provided by LIB500 *)
  C_En_DDS_0X401 : BOOL;  (* Message enable bit for message ID 16#401 *)
  S_SentOk_DDS_2_0X402 : BOOL;  (* Message sent status provided by LIB500 *)
  C_En_DDS_2_0X402 : BOOL;  (* Message enable bit for message ID 16#402 *)
  S_SentOk_HV_Durum_0X450 : BOOL;  (* Message sent status provided by LIB500 *)
  C_En_HV_Durum_0X450 : BOOL;  (* Message enable bit for message ID 16#450 *)
  S_SentOk_TCU_Trolleybus_Durum_0X460 : BOOL;  (* Message sent status provided by LIB500 *)
  S_SentOk_TCU_Ebus_Durum_0X461 : BOOL;  (* Message sent status provided by LIB500 *)
  C_En_TCU_Trolleybus_Durum_0X460 : BOOL;  (* Message enable bit for message ID 16#460 *)
  C_En_TCU_Ebus_Durum_0X461 : BOOL;  (* Message enable bit for message ID 16#461 *)
  S_SentOk_TCU_Surus_Limit_0X462 : BOOL;  (* Message sent status provided by LIB500 *)
  C_En_TCU_Surus_Limit_0X462 : BOOL;  (* Message enable bit for message ID 16#462 *)
  S_SentOk_TCU_Analog_0X463 : BOOL;  (* Message sent status provided by LIB500 *)
  C_En_TCU_Analog_0X463 : BOOL;  (* Message enable bit for message ID 16#463 *)
  S_SentOk_TCU_Cikis_Akim_Guc_0X464 : BOOL;  (* Message sent status provided by LIB500 *)
  C_En_TCU_Cikis_Akim_Guc_0X464 : BOOL;  (* Message enable bit for message ID 16#464 *)
  S_SentOk_TCU_Tork_Hiz_0X465 : BOOL;  (* Message sent status provided by LIB500 *)
  C_En_TCU_Tork_Hiz_0X465 : BOOL;  (* Message enable bit for message ID 16#465 *)
  S_SentOk_TCU_Calisma_Suresi_0X466 : BOOL;  (* Message sent status provided by LIB500 *)
  C_En_TCU_Calisma_Suresi_0X466 : BOOL;  (* Message enable bit for message ID 16#466 *)
  S_SentOk_TCU_Analog_2_0X467 : BOOL;  (* Message sent status provided by LIB500 *)
  C_En_TCU_Analog_2_0X467 : BOOL;  (* Message enable bit for message ID 16#467 *)
  S_SentOk_Yardimci_Konvertor_Durum_0X480 : BOOL;  (* Message sent status provided by LIB500 *)
  C_En_Yardimci_Konvertor_Durum_0X480 : BOOL;  (* Message enable bit for message ID 16#480 *)
  S_SentOk_Yardimci_Konvertor_Akim_0X481 : BOOL;  (* Message sent status provided by LIB500 *)
  C_En_Yardimci_Konvertor_Akim_0X481 : BOOL;  (* Message enable bit for message ID 16#481 *)
  S_SentOk_Yardimci_Konvertor_Guc_0X482 : BOOL;  (* Message sent status provided by LIB500 *)
  C_En_Yardimci_Konvertor_Guc_0X482 : BOOL;  (* Message enable bit for message ID 16#482 *)
  S_SentOk_Batarya_Konvertor_Analog_0X483 : BOOL;
  C_En_Batarya_Sarj_Konvertor_Analog_0X483 : BOOL;  (* Message enable bit for message ID 16#483 *)
  S_SentOk_Yardimci_Konvertor_Sicaklik_0X484 : BOOL;  (* Message sent status provided by LIB500 *)
  C_En_Yardimci_Konvertor_Sicaklik_0X484 : BOOL;  (* Message enable bit for message ID 16#484 *)
  S_SentOk_Isolation_Status_0X485 : BOOL;  (* Message sent status provided by LIB500 *)
  C_En_Isolation_Status_0X485 : BOOL;  (* Message enable bit for message ID 16#485 *)
  S_SentOk_Arac_Genel_Istatistik_0X4C2 : BOOL;  (* Message sent status provided by LIB500 *)
  C_En_Arac_Genel_Istatistik_0X4C2 : BOOL;  (* Message enable bit for message ID 16#4C2 *)
  S_SentOk_Temel_Durum_0X99 : BOOL;  (* Message sent status provided by LIB500 *)
  C_En_Temel_Durum_0X99 : BOOL;  (* Message enable bit for message ID 16#99 *)
  S_SentOk_ESS_Durum_0X430 : BOOL;  (* Message sent status provided by LIB500 *)
  C_En_ESS_Durum_0X430 : BOOL;  (* Message enable bit for message ID 16#430 *)
  S_SentOk_ESS_Paket_Voltaji_0X431 : BOOL;  (* Message sent status provided by LIB500 *)
  C_En_ESS_Paket_Voltaji_0X431 : BOOL;  (* Message enable bit for message ID 16#431 *)
  S_SentOk_ESS_Paket_Akim_0X432 : BOOL;  (* Message sent status provided by LIB500 *)
  C_En_ESS_Paket_Akim_0X432 : BOOL;  (* Message enable bit for message ID 16#432 *)
  S_SentOk_ESS_Maksimum_Hucre_Voltaji_0X433 : BOOL;  (* Message sent status provided by LIB500 *)
  C_En_ESS_Maksimum_Hucre_Voltaji_0X433 : BOOL;  (* Message enable bit for message ID 16#433 *)
  S_SentOk_ESS_Minimum_Hucre_Voltaji_0X434 : BOOL;  (* Message sent status provided by LIB500 *)
  C_En_ESS_Minimum_Hucre_Voltaji_0X434 : BOOL;  (* Message enable bit for message ID 16#434 *)
  S_SentOk_ESS_Ortalama_Hucre_Voltaji_0X435 : BOOL;  (* Message sent status provided by LIB500 *)
  C_En_ESS_Ortalama_Hucre_Voltaji_0X435 : BOOL;  (* Message enable bit for message ID 16#435 *)
  S_SentOk_ESS_Sicaklik_0X436 : BOOL;  (* Message sent status provided by LIB500 *)
  C_En_ESS_Sicaklik_0X436 : BOOL;  (* Message enable bit for message ID 16#436 *)
  S_SentOk_ESS_Analog_0X437 : BOOL;  (* Message sent status provided by LIB500 *)
  C_En_ESS_Analog_0X437 : BOOL;  (* Message enable bit for message ID 16#437 *)
  S_SentOk_ESS_Sogutma_Suyu_0X438 : BOOL;  (* Message sent status provided by LIB500 *)
  C_En_ESS_Sogutma_Suyu_0X438 : BOOL;  (* Message enable bit for message ID 16#438 *)
  S_SentOk_Sarj_Durum_0X4A0 : BOOL;  (* Message sent status provided by LIB500 *)
  C_En_Sarj_Durum_0X4A0 : BOOL;  (* Message enable bit for message ID 16#4A0 *)
  S_SentOk_Sarj_Sureleri_0X4A5 : BOOL;  (* Message sent status provided by LIB500 *)
  C_En_Sarj_Sureleri_0X4A5 : BOOL;  (* Message enable bit for message ID 16#4A5 *)
  S_SentOk_Sarj_Durum_3_0X4A6 : BOOL;  (* Message sent status provided by LIB500 *)
  C_En_Sarj_Durum_3_0X4A6 : BOOL;  (* Message enable bit for message ID 16#4A6 *)
  S_SentOk_Pantograph_Analog_4_0X4AF : BOOL;  (* Message sent status provided by LIB500 *)
  C_En_Pantograph_Analog_4_0X4AF : BOOL;  (* Message enable bit for message ID 16#4AF *)
  S_SentOk_Left_Charge_Analog_1_0X4B0 : BOOL;  (* Message sent status provided by LIB500 *)
  C_En_Left_Charge_Analog_1_0X4B0 : BOOL;  (* Message enable bit for message ID 16#4B0 *)
  S_SentOk_Hava_Kompresoru_Durum_0X4F0 : BOOL;  (* Message sent status provided by LIB500 *)
  C_En_Hava_Kompresoru_Durum_0X4F0 : BOOL;  (* Message enable bit for message ID 16#4F0 *)
  S_SentOk_ECU_Parametre_0X403 : BOOL;  (* Message sent status provided by LIB500 *)
  C_En_ECU_Parametre_0X403 : BOOL;  (* Message enable bit for message ID 16#403 *)
  S_SentOk_HVAC_Durum_0X410 : BOOL;  (* Message sent status provided by LIB500 *)
  C_En_HVAC_Durum_0X410 : BOOL;  (* Message enable bit for message ID 16#410 *)
  S_SentOk_HVAC_Sicaklik_0X411 : BOOL;  (* Message sent status provided by LIB500 *)
  C_En_HVAC_Sicaklik_0X411 : BOOL;  (* Message enable bit for message ID 16#411 *)
  S_SentOk_HVAC_Analog_0X413 : BOOL;  (* Message sent status provided by LIB500 *)
  C_En_HVAC_Analog_0X413 : BOOL;  (* Message enable bit for message ID 16#413 *)
  S_SentOk_Klima_Kontaktor_Kontrol_0X414 : BOOL;  (* Message sent status provided by LIB500 *)
  C_En_Klima_Kontaktor_Kontrol_0X414 : BOOL;  (* Message enable bit for message ID 16#414 *)
  S_SentOk_HVAC_Parameters_1_0X415 : BOOL;  (* Message sent status provided by LIB500 *)
  C_En_HVAC_Parameters_1_0X415 : BOOL;  (* Message enable bit for message ID 16#403 *)
  S_SentOk_HVAC_Water_Temperature_0X416 : BOOL;  (* Message sent status provided by LIB500 *)
  C_En_HVAC_Water_Temperature_0X416 : BOOL;  (* Message enable bit for message ID 16#403 *)
  S_SentOk_Arac_Menzil_0X4C0 : BOOL;  (* Message sent status provided by LIB500 *)
  C_En_Arac_Menzil_0X4C0 : BOOL;  (* Message enable bit for message ID 16#4C0 *)
  S_SentOk_Arac_Odometre_0X4C1 : BOOL;  (* Message sent status provided by LIB500 *)
  C_En_Arac_Odometre_0X4C1 : BOOL;  (* Message enable bit for message ID 16#4C1 *)
  S_SentOk_Arac_Surus_Enerji_0X4C3 : BOOL;  (* Message sent status provided by LIB500 *)
  C_En_Arac_Surus_Enerji_0X4C3 : BOOL;  (* Message enable bit for message ID 16#4C3 *)
  S_SentOk_Arac_Tuketilen_Enerji_1_0X4C4 : BOOL;  (* Message sent status provided by LIB500 *)
  C_En_Arac_Tuketilen_Enerji_1_0X4C4 : BOOL;  (* Message enable bit for message ID 16#4C4 *)
  S_SentOk_Arac_Tuketilen_Enerji_2_0X4C5 : BOOL;  (* Message sent status provided by LIB500 *)
  C_En_Arac_Tuketilen_Enerji_2_0X4C5 : BOOL;  (* Message enable bit for message ID 16#4C5 *)
  S_SentOk_Arac_Kapasite_0X4C6 : BOOL;  (* Message sent status provided by LIB500 *)
  C_En_Arac_Kapasite_0X4C6 : BOOL;  (* Message enable bit for message ID 16#4C6 *)
  S_SentOk_Arac_Sureler_0X4C7 : BOOL;  (* Message sent status provided by LIB500 *)
  C_En_Arac_Sureler_0X4C7 : BOOL;  (* Message enable bit for message ID 16#4C7 *)
  S_SentOk_Arac_Toplam_Tuketilen_Enerji_0X4C8 : BOOL;  (* Message sent status provided by LIB500 *)
  C_En_Arac_Toplam_Tuketilen_Enerji_0X4C8 : BOOL;  (* Message enable bit for message ID 16#4C8 *)
  S_SentOk_Arac_Genel_Istatistik_2_0X4C9 : BOOL;  (* Message sent status provided by LIB500 *)
  C_En_Arac_Genel_Istatistik_2_0X4C9 : BOOL;  (* Message enable bit for message ID 16#4C9 *)
  S_SentOk_Klima_Calisma_Sureleri_1_0X4CA : BOOL;  (* Message sent status provided by LIB500 *)
  C_En_Klima_Calisma_Sureleri_1_0X4CA : BOOL;  (* Message enable bit for message ID 16#4CA *)
  S_SentOk_Klima_Calisma_Sureleri_2_0X4CB : BOOL;  (* Message sent status provided by LIB500 *)
  C_En_Klima_Calisma_Sureleri_2_0X4CB : BOOL;  (* Message enable bit for message ID 16#4CB *)
  S_SentOk_Sayicilar_1_0X4CC : BOOL;  (* Message sent status provided by LIB500 *)
  C_En_Sayicilar_1_0X4CC : BOOL;  (* Message enable bit for message ID 16#4CC *)
  S_SentOk_Yardimci_Tuketici_Enerjileri_0X4CD : BOOL;  (* Message sent status provided by LIB500 *)
  C_En_Yardimci_Tuketici_Enerjileri_0X4CD : BOOL;  (* Message enable bit for message ID 16#4CD *)
  S_SentOk_Kapi_Sayicilari_1_0X4CE : BOOL;  (* Message sent status provided by LIB500 *)
  C_En_Kapi_Sayicilari_1_0X4CE : BOOL;  (* Message enable bit for message ID 16#4CD *)
  S_SentOk_Kapi_Sayicilari_2_0X4CF : BOOL;  (* Message sent status provided by LIB500 *)
  C_En_Kapi_Sayicilari_2_0X4CF : BOOL;  (* Message enable bit for message ID 16#4CE *)
  S_SentOk_Sarj_Enerjisi_0X4D0 : BOOL;  (* Message sent status provided by LIB500 *)
  C_En_Sarj_Enerjisi_0X4D0 : BOOL;  (* Message enable bit for message ID 16#4CF *)
  S_SentOk_Arac_Bilgi_1_0X4E0 : BOOL;  (* Message sent status provided by LIB500 *)
  C_En_Arac_Bilgi_1_0X4E0 : BOOL;  (* Message enable bit for message ID 16#4E0 *)
  S_SentOk_Arac_Bilgi_2_0X4E1 : BOOL;  (* Message sent status provided by LIB500 *)
  C_En_Arac_Bilgi_2_0X4E1 : BOOL;  (* Message enable bit for message ID 16#4E1 *)
  S_SentOk_Olay_Durum_0X500 : BOOL;  (* Message sent status provided by LIB500 *)
  C_En_Olay_Durum_0X500 : BOOL;  (* Message enable bit for message ID 16#500 *)
END_STRUCT;
END_TYPE

TYPE IC_T : STRUCT
  S_Pwr_Stg : lib500_types.IO_POWER_STATUS;  (* System Status *)
  S_Sfty_Swc_0 : lib500_types.IO_POWER_STATUS;
  S_Sfty_Swc_1 : lib500_types.IO_POWER_STATUS;
  S_Sfty_Swc_2 : lib500_types.IO_POWER_STATUS;
  S_Snsr_Sp_0 : lib500_types.IO_POWER_STATUS;
  S_Snsr_Sp_1 : lib500_types.IO_POWER_STATUS;
  S_Snsr_Sp_2 : lib500_types.IO_POWER_STATUS;
  S_Term15 : lib500_types.IO_POWER_STATUS;
  S_Wkup : lib500_types.IO_POWER_STATUS;
  C_ECU_Pwr : lib500_types.IO_POWER_STATE := lib500_types.IO_POWER_STATE.IO_POWER_OFF;  (* System Control *)
  C_Snsr_Sp : lib500_types.IO_POWER_STATE := lib500_types.IO_POWER_STATE.IO_POWER_OFF;
  C_Sfty_Swc : lib500_types.IO_POWER_STATE := lib500_types.IO_POWER_STATE.IO_POWER_OFF;
  S_Diag : lib500_types.DIAG_STATUS;  (* System Diagnostic *)
  X_U_Bat : lib500_types.IO_ADC_STATUS;  (* System Auxiliary Measurement *)
  X_U_Term15 : lib500_types.IO_ADC_STATUS;
  X_U_Wkup : lib500_types.IO_ADC_STATUS;
  X_T_ECU : lib500_types.IO_ADC_TEMPERATURE;  (* System Internal Measurement *)
  X_U_Sfty_Swc_0 : lib500_types.IO_ADC_STATUS;
  X_U_Sfty_Swc_1 : lib500_types.IO_ADC_STATUS;
  X_U_Sfty_Swc_2 : lib500_types.IO_ADC_STATUS;
  X_U_Snsr_Sp_0 : lib500_types.IO_ADC_STATUS;
  X_U_Snsr_Sp_1 : lib500_types.IO_ADC_STATUS;
  X_U_Snsr_Sp_2 : lib500_types.IO_ADC_STATUS;
  Obj_CAN0 : tCan;  (* DIAG CAN - Bozankaya Diag, ATS *)
  Obj_CAN1 : tCan;  (* PCAN - VCU, TCU, EBS, Steering Angle Sensor, ACU, Pantograph *)
  Obj_CAN2 : tCan;  (* TCU CAN - TCU *)
  Obj_CAN3 : tCan;  (* TRDU CAN - TRDU *)
  Obj_CAN5 : tCan;  (* BMS CAN - BMS *)
  Obj_CAN6 : tCan;  (* AC CAN - HVAC *)
  S_Diag_CAN_En_Cnt : INT;
  S_Diag_250ms_Actv : BOOL;
  S_Diag_500ms_Actv : BOOL;
  S_Diag_1000ms_Actv : BOOL;
  X_Sw_Ver_Mjr_ECU : REAL;  (* ECU SW VERSION *)
  X_Sw_Ver_Mnr_ECU : REAL;
  X_Sw_Ver_Tst_ECU : REAL;
  S_Err_Sw_Ver : BOOL := FALSE;
  X_Prj_No : WORD;
END_STRUCT;
END_TYPE

(* Added BY Deniz Çıkış, @16.10.2023 *)
TYPE Param_T : STRUCT
  X_No : BYTE;
  X_Val : REAL;
  X_Usr_Id : BYTE;
  X_Seconds : BYTE;
  X_Minutes : BYTE;
  X_Hours : BYTE;
  X_Days : BYTE;
  X_Months : BYTE;
  X_Years : BYTE;
END_STRUCT;
END_TYPE

FUNCTION_BLOCK _FB_CanRx_Message
  VAR_INPUT
    C_Enable : BOOL := FALSE;  (* Enable message *)
    Obj_CAN : POINTER TO tCan;  (* CAN Object derived from CAN_500_LIB *)
    X_MsgID : UDINT := 0;  (* Message ID *)
    Tm_MsgTmOut : TIME := TIME#500ms;  (* Message time limit *)
    S_Extended : BOOL := FALSE;  (* Message extended bit *)
  END_VAR
  VAR_OUTPUT
    S_ER_TmOut : BOOL;  (* Input data endpoints *)
    X_Byte_0 : BYTE;  (* Input data endpoints *)
    X_Byte_1 : BYTE;  (* Input data endpoints *)
    X_Byte_2 : BYTE;  (* Input data endpoints *)
    X_Byte_3 : BYTE;  (* Input data endpoints *)
    X_Byte_4 : BYTE;  (* Input data endpoints *)
    X_Byte_5 : BYTE;  (* Input data endpoints *)
    X_Byte_6 : BYTE;  (* Input data endpoints *)
    X_Byte_7 : BYTE;  (* Input data endpoints *)
  END_VAR
  VAR
    fb_message : CanRx;  (* Library object container *)
  END_VAR

                    
(*
**********************************************************************
Bozankaya A.Ş.
**********************************************************************
Name					: _FB_CanRx_Message
POU Type				: FB
Created by 				: E.TURKER , BZK.
Creation Date 			: 09-03-2022
Modifications			: see version description below


FB Description:
This FB handles the RX can messages according to CAN_500_LIB
*********************************************************************

